LIN {X 0,Y 369.464,Z 431.864,A -85,B 0,C 180,E1 -12702.078,E2 -12702.078} C_VEL
LIN {X 0,Y 369.996,Z 423.683,A -85,B 0,C 180,E1 -12702.896,E2 -12702.896} C_VEL
LIN {X 0,Y 370.537,Z 415.209,A -85,B 0,C 180,E1 -12703.575,E2 -12703.575} C_VEL
LIN {X 0,Y 371.025,Z 406.559,A -85,B 0,C 180,E1 -12704.116,E2 -12704.116} C_VEL
LIN {X 0,Y 371.546,Z 395.482,A -85,B 0,C 180,E1 -12704.62,E2 -12704.62} C_VEL
LIN {X 0,Y 371.88,Z 379.251,A -85,B 0,C 180,E1 -12705.026,E2 -12705.026} C_VEL
LIN {X 0,Y 372.213,Z 341.609,A -85,B 0,C 180,E1 -12705.819,E2 -12705.819} C_VEL
LIN {X 0,Y 369.031,Z 313.014,A -85,B 0,C 180,E1 -12706.559,E2 -12706.559} C_VEL
LIN {X 0,Y 370.022,Z 297.413,A -85,B 0,C 180,E1 -12710.281,E2 -12710.281} C_VEL
LIN {X 0,Y 371.123,Z 283.099,A -85,B 0,C 180,E1 -12713.729,E2 -12713.729} C_VEL
LIN {X 0,Y 370.607,Z 278.235,A -85,B 0,C 180,E1 -12714.957,E2 -12714.957} C_VEL
LIN {X 0,Y 369.016,Z 269.333,A -85,B 0,C 180,E1 -12717.276,E2 -12717.276} C_VEL
LIN {X 0,Y 368.912,Z 269.342,A -85,B 0,C 180,E1 -12720.987,E2 -12720.987} C_VEL
LIN {X 0,Y 368.937,Z 269.338,A -85,B 0,C 180,E1 -12724.853,E2 -12724.853} C_VEL
LIN {X 0,Y 368.909,Z 269.341,A -85,B 0,C 180,E1 -12728.64,E2 -12728.64} C_VEL
LIN {X 0,Y 368.881,Z 269.346,A -85,B 0,C 180,E1 -12732.009,E2 -12732.009} C_VEL
LIN {X 0,Y 368.879,Z 269.347,A -85,B 0,C 180,E1 -12735.175,E2 -12735.175} C_VEL
LIN {X 0,Y 368.881,Z 269.345,A -85,B 0,C 180,E1 -12738.177,E2 -12738.177} C_VEL
LIN {X 0,Y 368.906,Z 269.346,A -85,B 0,C 180,E1 -12741.359,E2 -12741.359} C_VEL
LIN {X 0,Y 368.935,Z 269.34,A -85,B 0,C 180,E1 -12745.146,E2 -12745.146} C_VEL
LIN {X 0,Y 368.928,Z 269.34,A -85,B 0,C 180,E1 -12749.046,E2 -12749.046} C_VEL
LIN {X 0,Y 368.977,Z 269.339,A -85,B 0,C 180,E1 -12751.563,E2 -12751.563} C_VEL
LIN {X 0,Y 368.997,Z 269.332,A -85,B 0,C 180,E1 -12754.019,E2 -12754.019} C_VEL
LIN {X 0,Y 368.929,Z 269.345,A -85,B 0,C 180,E1 -12757.604,E2 -12757.604} C_VEL
LIN {X 0,Y 368.963,Z 269.336,A -85,B 0,C 180,E1 -12761.105,E2 -12761.105} C_VEL
LIN {X 0,Y 368.994,Z 269.33,A -85,B 0,C 180,E1 -12764.534,E2 -12764.534} C_VEL
LIN {X 0,Y 369.001,Z 269.333,A -85,B 0,C 180,E1 -12767.906,E2 -12767.906} C_VEL
LIN {X 0,Y 369.162,Z 269.313,A -85,B 0,C 180,E1 -12771.868,E2 -12771.868} C_VEL
LIN {X 0,Y 369.139,Z 269.313,A -85,B 0,C 180,E1 -12774.537,E2 -12774.537} C_VEL
LIN {X 0,Y 369.313,Z 269.295,A -85,B 0,C 180,E1 -12777.818,E2 -12777.818} C_VEL
LIN {X 0,Y 369.453,Z 269.276,A -85,B 0,C 180,E1 -12779.999,E2 -12779.999} C_VEL
LIN {X 0,Y 369.313,Z 269.292,A -85,B 0,C 180,E1 -12782.18,E2 -12782.18} C_VEL
LIN {X 0,Y 369.197,Z 269.305,A -85,B 0,C 180,E1 -12786.628,E2 -12786.628} C_VEL
LIN {X 0,Y 369.133,Z 269.313,A -85,B 0,C 180,E1 -12788.76,E2 -12788.76} C_VEL
LIN {X 0,Y 369.006,Z 269.331,A -85,B 0,C 180,E1 -12792.092,E2 -12792.092} C_VEL
LIN {X 0,Y 368.992,Z 269.335,A -85,B 0,C 180,E1 -12795.464,E2 -12795.464} C_VEL
LIN {X 0,Y 368.983,Z 269.332,A -85,B 0,C 180,E1 -12798.892,E2 -12798.892} C_VEL
LIN {X 0,Y 368.93,Z 269.339,A -85,B 0,C 180,E1 -12802.394,E2 -12802.394} C_VEL
LIN {X 0,Y 368.992,Z 269.334,A -85,B 0,C 180,E1 -12805.979,E2 -12805.979} C_VEL
LIN {X 0,Y 368.907,Z 269.348,A -85,B 0,C 180,E1 -12809.69,E2 -12809.69} C_VEL
LIN {X 0,Y 368.889,Z 269.345,A -85,B 0,C 180,E1 -12813.042,E2 -12813.042} C_VEL
LIN {X 0,Y 368.91,Z 269.343,A -85,B 0,C 180,E1 -12816.196,E2 -12816.196} C_VEL
LIN {X 0,Y 368.899,Z 269.343,A -85,B 0,C 180,E1 -12818.952,E2 -12818.952} C_VEL
LIN {X 0,Y 368.901,Z 269.345,A -85,B 0,C 180,E1 -12822.014,E2 -12822.014} C_VEL
LIN {X 0,Y 368.946,Z 269.338,A -85,B 0,C 180,E1 -12825.187,E2 -12825.187} C_VEL
LIN {X 0,Y 368.937,Z 269.34,A -85,B 0,C 180,E1 -12828.186,E2 -12828.186} C_VEL
LIN {X 0,Y 368.904,Z 269.345,A -85,B 0,C 180,E1 -12831.358,E2 -12831.358} C_VEL
LIN {X 0,Y 368.928,Z 269.34,A -85,B 0,C 180,E1 -12835.146,E2 -12835.146} C_VEL
LIN {X 0,Y 368.921,Z 269.34,A -85,B 0,C 180,E1 -12839.046,E2 -12839.046} C_VEL
LIN {X 0,Y 368.971,Z 269.338,A -85,B 0,C 180,E1 -12841.564,E2 -12841.564} C_VEL
LIN {X 0,Y 368.991,Z 269.334,A -85,B 0,C 180,E1 -12844.019,E2 -12844.019} C_VEL
LIN {X 0,Y 368.925,Z 269.344,A -85,B 0,C 180,E1 -12847.605,E2 -12847.605} C_VEL
LIN {X 0,Y 368.975,Z 269.334,A -85,B 0,C 180,E1 -12851.107,E2 -12851.107} C_VEL
LIN {X 0,Y 368.989,Z 269.332,A -85,B 0,C 180,E1 -12854.535,E2 -12854.535} C_VEL
LIN {X 0,Y 368.997,Z 269.335,A -85,B 0,C 180,E1 -12857.906,E2 -12857.906} C_VEL
LIN {X 0,Y 369.22,Z 269.308,A -85,B 0,C 180,E1 -12861.801,E2 -12861.801} C_VEL
LIN {X 0,Y 369.133,Z 269.314,A -85,B 0,C 180,E1 -12864.537,E2 -12864.537} C_VEL
LIN {X 0,Y 369.307,Z 269.297,A -85,B 0,C 180,E1 -12867.819,E2 -12867.819} C_VEL
LIN {X 0,Y 369.449,Z 269.278,A -85,B 0,C 180,E1 -12870,E2 -12870} C_VEL
LIN {X 0,Y 369.307,Z 269.294,A -85,B 0,C 180,E1 -12872.181,E2 -12872.181} C_VEL
LIN {X 0,Y 369.189,Z 269.307,A -85,B 0,C 180,E1 -12876.558,E2 -12876.558} C_VEL
LIN {X 0,Y 369.113,Z 269.316,A -85,B 0,C 180,E1 -12878.761,E2 -12878.761} C_VEL
LIN {X 0,Y 369.003,Z 269.333,A -85,B 0,C 180,E1 -12882.093,E2 -12882.093} C_VEL
LIN {X 0,Y 368.989,Z 269.334,A -85,B 0,C 180,E1 -12885.465,E2 -12885.465} C_VEL
LIN {X 0,Y 368.948,Z 269.337,A -85,B 0,C 180,E1 -12888.894,E2 -12888.894} C_VEL
LIN {X 0,Y 368.915,Z 269.342,A -85,B 0,C 180,E1 -12892.395,E2 -12892.395} C_VEL
LIN {X 0,Y 368.989,Z 269.336,A -85,B 0,C 180,E1 -12895.98,E2 -12895.98} C_VEL
LIN {X 0,Y 368.909,Z 269.346,A -85,B 0,C 180,E1 -12899.69,E2 -12899.69} C_VEL
LIN {X 0,Y 368.983,Z 269.414,A -85,B 0,C 180,E1 -12901.322,E2 -12901.322} C_VEL
LIN {X 0,Y 369.531,Z 273.509,A -85,B 0,C 180,E1 -12902.538,E2 -12902.538} C_VEL
LIN {X 0,Y 372.803,Z 292.013,A -85,B 0,C 180,E1 -12903.079,E2 -12903.079} C_VEL
LIN {X 0,Y 372.124,Z 332.295,A -85,B 0,C 180,E1 -12903.917,E2 -12903.917} C_VEL
LIN {X 0,Y 371.303,Z 338.133,A -85,B 0,C 180,E1 -12904.01,E2 -12904.01} C_VEL
LIN {X 0,Y 365.612,Z 355.514,A -85,B 0,C 180,E1 -12904.276,E2 -12904.276} C_VEL
LIN {X 0,Y 364.732,Z 360.703,A -85,B 0,C 180,E1 -12904.47,E2 -12904.47} C_VEL
LIN {X 0,Y 364.647,Z 362.591,A -85,B 0,C 180,E1 -12904.557,E2 -12904.557} C_VEL
LIN {X 0,Y 364.216,Z 373.541,A -85,B 0,C 180,E1 -12905.21,E2 -12905.21} C_VEL
LIN {X 0,Y 363.762,Z 382.837,A -85,B 0,C 180,E1 -12905.955,E2 -12905.955} C_VEL
LIN {X 0,Y 363.399,Z 390.285,A -85,B 0,C 180,E1 -12906.699,E2 -12906.699} C_VEL
LIN {X 0,Y 362.909,Z 397.891,A -85,B 0,C 180,E1 -12907.62,E2 -12907.62} C_VEL
LIN {X 0,Y 362.404,Z 404.176,A -85,B 0,C 180,E1 -12908.532,E2 -12908.532} C_VEL
LIN {X 0,Y 361.95,Z 410.539,A -85,B 0,C 180,E1 -12909.642,E2 -12909.642} C_VEL
LIN {X 0,Y 361.646,Z 415.686,A -85,B 0,C 180,E1 -12910.723,E2 -12910.723} C_VEL
LIN {X 0,Y 361.224,Z 420.228,A -85,B 0,C 180,E1 -12911.862,E2 -12911.862} C_VEL
LIN {X 0,Y 360.948,Z 425.143,A -85,B 0,C 180,E1 -12913.423,E2 -12913.423} C_VEL
LIN {X 0,Y 360.756,Z 427.858,A -85,B 0,C 180,E1 -12914.532,E2 -12914.532} C_VEL
LIN {X 0,Y 360.592,Z 429.716,A -85,B 0,C 180,E1 -12915.443,E2 -12915.443} C_VEL
LIN {X 0,Y 360.403,Z 431.851,A -85,B 0,C 180,E1 -12916.962,E2 -12916.962} C_VEL
LIN {X 0,Y 360.327,Z 433.016,A -85,B 0,C 180,E1 -12918.461,E2 -12918.461} C_VEL
LIN {X 0,Y 360.394,Z 433.266,A -85,B 0,C 180,E1 -12919.946,E2 -12919.946} C_VEL
LIN {X 0,Y 360.52,Z 432.637,A -85,B 0,C 180,E1 -12921.407,E2 -12921.407} C_VEL
LIN {X 0,Y 360.787,Z 430.932,A -85,B 0,C 180,E1 -12923.001,E2 -12923.001} C_VEL
LIN {X 0,Y 361.041,Z 428.802,A -85,B 0,C 180,E1 -12924.271,E2 -12924.271} C_VEL
LIN {X 0,Y 361.424,Z 425.566,A -85,B 0,C 180,E1 -12925.675,E2 -12925.675} C_VEL
LIN {X 0,Y 362.019,Z 420.207,A -85,B 0,C 180,E1 -12927.405,E2 -12927.405} C_VEL
LIN {X 0,Y 362.647,Z 414.276,A -85,B 0,C 180,E1 -12928.862,E2 -12928.862} C_VEL
LIN {X 0,Y 363.301,Z 407.451,A -85,B 0,C 180,E1 -12930.172,E2 -12930.172} C_VEL
LIN {X 0,Y 364.05,Z 400.148,A -85,B 0,C 180,E1 -12931.302,E2 -12931.302} C_VEL
LIN {X 0,Y 364.715,Z 393.335,A -85,B 0,C 180,E1 -12932.174,E2 -12932.174} C_VEL
LIN {X 0,Y 365.239,Z 385.966,A -85,B 0,C 180,E1 -12932.962,E2 -12932.962} C_VEL
LIN {X 0,Y 365.741,Z 377.497,A -85,B 0,C 180,E1 -12933.695,E2 -12933.695} C_VEL
LIN {X 0,Y 366.277,Z 369.067,A -85,B 0,C 180,E1 -12934.264,E2 -12934.264} C_VEL
LIN {X 0,Y 366.592,Z 359.77,A -85,B 0,C 180,E1 -12934.742,E2 -12934.742} C_VEL
LIN {X 0,Y 366.828,Z 350.382,A -85,B 0,C 180,E1 -12935.072,E2 -12935.072} C_VEL
LIN {X 0,Y 367.979,Z 292.659,A -85,B 0,C 180,E1 -12936.356,E2 -12936.356} C_VEL
LIN {X 0,Y 365.505,Z 281.786,A -85,B 0,C 180,E1 -12936.768,E2 -12936.768} C_VEL
LIN {X 0,Y 362.818,Z 274.529,A -85,B 0,C 180,E1 -12937.132,E2 -12937.132} C_VEL
LIN {X 0,Y 361.896,Z 270.225,A -85,B 0,C 180,E1 -12938.349,E2 -12938.349} C_VEL
LIN {X 0,Y 361.957,Z 270.215,A -85,B 0,C 180,E1 -12942.062,E2 -12942.062} C_VEL
LIN {X 0,Y 361.988,Z 270.207,A -85,B 0,C 180,E1 -12946.102,E2 -12946.102} C_VEL
LIN {X 0,Y 362.022,Z 270.202,A -85,B 0,C 180,E1 -12949.939,E2 -12949.939} C_VEL
LIN {X 0,Y 362.158,Z 270.185,A -85,B 0,C 180,E1 -12953.315,E2 -12953.315} C_VEL
LIN {X 0,Y 362.275,Z 270.166,A -85,B 0,C 180,E1 -12957.777,E2 -12957.777} C_VEL
LIN {X 0,Y 362.419,Z 270.153,A -85,B 0,C 180,E1 -12960.001,E2 -12960.001} C_VEL
LIN {X 0,Y 362.275,Z 270.17,A -85,B 0,C 180,E1 -12962.225,E2 -12962.225} C_VEL
LIN {X 0,Y 362.164,Z 270.185,A -85,B 0,C 180,E1 -12966.687,E2 -12966.687} C_VEL
LIN {X 0,Y 362.067,Z 270.194,A -85,B 0,C 180,E1 -12968.934,E2 -12968.934} C_VEL
LIN {X 0,Y 361.952,Z 270.205,A -85,B 0,C 180,E1 -12972.333,E2 -12972.333} C_VEL
LIN {X 0,Y 361.955,Z 270.212,A -85,B 0,C 180,E1 -12974.621,E2 -12974.621} C_VEL
LIN {X 0,Y 361.953,Z 270.207,A -85,B 0,C 180,E1 -12978.1,E2 -12978.1} C_VEL
LIN {X 0,Y 361.886,Z 270.211,A -85,B 0,C 180,E1 -12981.654,E2 -12981.654} C_VEL
LIN {X 0,Y 361.923,Z 270.205,A -85,B 0,C 180,E1 -12985.291,E2 -12985.291} C_VEL
LIN {X 0,Y 361.917,Z 270.214,A -85,B 0,C 180,E1 -12987.779,E2 -12987.779} C_VEL
LIN {X 0,Y 361.842,Z 270.223,A -85,B 0,C 180,E1 -12991.286,E2 -12991.286} C_VEL
LIN {X 0,Y 361.85,Z 270.218,A -85,B 0,C 180,E1 -12994.282,E2 -12994.282} C_VEL
LIN {X 0,Y 361.862,Z 270.216,A -85,B 0,C 180,E1 -12997.224,E2 -12997.224} C_VEL
LIN {X 0,Y 361.87,Z 270.218,A -85,B 0,C 180,E1 -13000.763,E2 -13000.763} C_VEL
LIN {X 0,Y 361.861,Z 270.22,A -85,B 0,C 180,E1 -13004.362,E2 -13004.362} C_VEL
LIN {X 0,Y 361.834,Z 270.225,A -85,B 0,C 180,E1 -13007.569,E2 -13007.569} C_VEL
LIN {X 0,Y 361.869,Z 270.221,A -85,B 0,C 180,E1 -13010.974,E2 -13010.974} C_VEL
LIN {X 0,Y 361.873,Z 270.223,A -85,B 0,C 180,E1 -13014.656,E2 -13014.656} C_VEL
LIN {X 0,Y 361.837,Z 270.228,A -85,B 0,C 180,E1 -13018.372,E2 -13018.372} C_VEL
LIN {X 0,Y 361.918,Z 270.267,A -85,B 0,C 180,E1 -13022.183,E2 -13022.183} C_VEL
LIN {X 0,Y 363.78,Z 279.211,A -85,B 0,C 180,E1 -13024.542,E2 -13024.542} C_VEL
LIN {X 0,Y 364.457,Z 284.393,A -85,B 0,C 180,E1 -13025.849,E2 -13025.849} C_VEL
LIN {X 0,Y 363.322,Z 299.23,A -85,B 0,C 180,E1 -13029.328,E2 -13029.328} C_VEL
LIN {X 0,Y 362.603,Z 310.337,A -85,B 0,C 180,E1 -13031.912,E2 -13031.912} C_VEL
LIN {X 0,Y 366.013,Z 332.015,A -85,B 0,C 180,E1 -13032.637,E2 -13032.637} C_VEL
LIN {X 0,Y 367.237,Z 345.692,A -85,B 0,C 180,E1 -13033.023,E2 -13033.023} C_VEL
LIN {X 0,Y 366.326,Z 389.941,A -85,B 0,C 180,E1 -13034.016,E2 -13034.016} C_VEL
LIN {X 0,Y 365.823,Z 401.663,A -85,B 0,C 180,E1 -13034.47,E2 -13034.47} C_VEL
LIN {X 0,Y 365.072,Z 412.017,A -85,B 0,C 180,E1 -13035.08,E2 -13035.08} C_VEL
LIN {X 0,Y 364.371,Z 420.792,A -85,B 0,C 180,E1 -13035.764,E2 -13035.764} C_VEL
LIN {X 0,Y 363.598,Z 429.21,A -85,B 0,C 180,E1 -13036.589,E2 -13036.589} C_VEL
LIN {X 0,Y 362.832,Z 437.203,A -85,B 0,C 180,E1 -13037.556,E2 -13037.556} C_VEL
LIN {X 0,Y 362.272,Z 443.836,A -85,B 0,C 180,E1 -13038.531,E2 -13038.531} C_VEL
LIN {X 0,Y 361.636,Z 450.167,A -85,B 0,C 180,E1 -13039.645,E2 -13039.645} C_VEL
LIN {X 0,Y 361.155,Z 455.45,A -85,B 0,C 180,E1 -13040.762,E2 -13040.762} C_VEL
LIN {X 0,Y 360.783,Z 460.854,A -85,B 0,C 180,E1 -13042.163,E2 -13042.163} C_VEL
LIN {X 0,Y 360.496,Z 465.95,A -85,B 0,C 180,E1 -13043.863,E2 -13043.863} C_VEL
LIN {X 0,Y 360.451,Z 469.439,A -85,B 0,C 180,E1 -13045.527,E2 -13045.527} C_VEL
LIN {X 0,Y 360.376,Z 471.138,A -85,B 0,C 180,E1 -13046.646,E2 -13046.646} C_VEL
LIN {X 0,Y 360.426,Z 472.224,A -85,B 0,C 180,E1 -13047.765,E2 -13047.765} C_VEL
LIN {X 0,Y 360.513,Z 472.804,A -85,B 0,C 180,E1 -13048.883,E2 -13048.883} C_VEL
LIN {X 0,Y 360.515,Z 472.899,A -85,B 0,C 180,E1 -13050,E2 -13050} C_VEL
LIN {X 0,Y 360.522,Z 472.509,A -85,B 0,C 180,E1 -13051.117,E2 -13051.117} C_VEL
LIN {X 0,Y 360.47,Z 471.553,A -85,B 0,C 180,E1 -13052.235,E2 -13052.235} C_VEL
LIN {X 0,Y 360.434,Z 469.062,A -85,B 0,C 180,E1 -13053.913,E2 -13053.913} C_VEL
LIN {X 0,Y 360.475,Z 466.715,A -85,B 0,C 180,E1 -13055.033,E2 -13055.033} C_VEL
LIN {X 0,Y 360.582,Z 461.895,A -85,B 0,C 180,E1 -13056.716,E2 -13056.716} C_VEL
LIN {X 0,Y 360.8,Z 456.651,A -85,B 0,C 180,E1 -13058.119,E2 -13058.119} C_VEL
LIN {X 0,Y 361.108,Z 451.511,A -85,B 0,C 180,E1 -13059.24,E2 -13059.24} C_VEL
LIN {X 0,Y 361.499,Z 445.309,A -85,B 0,C 180,E1 -13060.36,E2 -13060.36} C_VEL
LIN {X 0,Y 361.896,Z 438.787,A -85,B 0,C 180,E1 -13061.34,E2 -13061.34} C_VEL
LIN {X 0,Y 362.509,Z 430.909,A -85,B 0,C 180,E1 -13062.313,E2 -13062.313} C_VEL
LIN {X 0,Y 363.057,Z 422.603,A -85,B 0,C 180,E1 -13063.147,E2 -13063.147} C_VEL
LIN {X 0,Y 363.66,Z 412.069,A -85,B 0,C 180,E1 -13063.979,E2 -13063.979} C_VEL
LIN {X 0,Y 364.264,Z 400.977,A -85,B 0,C 180,E1 -13064.593,E2 -13064.593} C_VEL
LIN {X 0,Y 364.685,Z 391.599,A -85,B 0,C 180,E1 -13064.947,E2 -13064.947} C_VEL
LIN {X 0,Y 365.233,Z 356.793,A -85,B 0,C 180,E1 -13065.725,E2 -13065.725} C_VEL
LIN {X 0,Y 365.323,Z 342.507,A -85,B 0,C 180,E1 -13066.035,E2 -13066.035} C_VEL
LIN {X 0,Y 362.032,Z 312.562,A -85,B 0,C 180,E1 -13066.849,E2 -13066.849} C_VEL
LIN {X 0,Y 362.985,Z 298.012,A -85,B 0,C 180,E1 -13070.396,E2 -13070.396} C_VEL
LIN {X 0,Y 364.132,Z 283.685,A -85,B 0,C 180,E1 -13073.911,E2 -13073.911} C_VEL
LIN {X 0,Y 363.095,Z 276.349,A -85,B 0,C 180,E1 -13075.817,E2 -13075.817} C_VEL
LIN {X 0,Y 361.958,Z 270.213,A -85,B 0,C 180,E1 -13077.454,E2 -13077.454} C_VEL
LIN {X 0,Y 361.848,Z 270.224,A -85,B 0,C 180,E1 -13081.285,E2 -13081.285} C_VEL
LIN {X 0,Y 361.855,Z 270.22,A -85,B 0,C 180,E1 -13084.28,E2 -13084.28} C_VEL
LIN {X 0,Y 361.871,Z 270.221,A -85,B 0,C 180,E1 -13087.224,E2 -13087.224} C_VEL
LIN {X 0,Y 361.836,Z 270.222,A -85,B 0,C 180,E1 -13090.755,E2 -13090.755} C_VEL
LIN {X 0,Y 361.816,Z 270.225,A -85,B 0,C 180,E1 -13094.368,E2 -13094.368} C_VEL
LIN {X 0,Y 361.835,Z 270.229,A -85,B 0,C 180,E1 -13097.567,E2 -13097.567} C_VEL
LIN {X 0,Y 361.867,Z 270.219,A -85,B 0,C 180,E1 -13100.973,E2 -13100.973} C_VEL
LIN {X 0,Y 361.873,Z 270.217,A -85,B 0,C 180,E1 -13104.654,E2 -13104.654} C_VEL
LIN {X 0,Y 361.837,Z 270.222,A -85,B 0,C 180,E1 -13108.37,E2 -13108.37} C_VEL
LIN {X 0,Y 361.899,Z 270.215,A -85,B 0,C 180,E1 -13110.954,E2 -13110.954} C_VEL
LIN {X 0,Y 361.952,Z 270.213,A -85,B 0,C 180,E1 -13113.474,E2 -13113.474} C_VEL
LIN {X 0,Y 361.887,Z 270.218,A -85,B 0,C 180,E1 -13117.144,E2 -13117.144} C_VEL
LIN {X 0,Y 361.908,Z 270.213,A -85,B 0,C 180,E1 -13120.723,E2 -13120.723} C_VEL
LIN {X 0,Y 361.93,Z 270.212,A -85,B 0,C 180,E1 -13123.065,E2 -13123.065} C_VEL
LIN {X 0,Y 361.995,Z 270.202,A -85,B 0,C 180,E1 -13126.527,E2 -13126.527} C_VEL
LIN {X 0,Y 362.027,Z 270.201,A -85,B 0,C 180,E1 -13129.937,E2 -13129.937} C_VEL
LIN {X 0,Y 362.158,Z 270.185,A -85,B 0,C 180,E1 -13133.313,E2 -13133.313} C_VEL
LIN {X 0,Y 362.277,Z 270.172,A -85,B 0,C 180,E1 -13137.776,E2 -13137.776} C_VEL
LIN {X 0,Y 362.422,Z 270.152,A -85,B 0,C 180,E1 -13139.999,E2 -13139.999} C_VEL
LIN {X 0,Y 362.277,Z 270.168,A -85,B 0,C 180,E1 -13142.223,E2 -13142.223} C_VEL
LIN {X 0,Y 362.166,Z 270.181,A -85,B 0,C 180,E1 -13146.685,E2 -13146.685} C_VEL
LIN {X 0,Y 362.07,Z 270.194,A -85,B 0,C 180,E1 -13148.932,E2 -13148.932} C_VEL
LIN {X 0,Y 361.96,Z 270.208,A -85,B 0,C 180,E1 -13152.331,E2 -13152.331} C_VEL
LIN {X 0,Y 361.956,Z 270.207,A -85,B 0,C 180,E1 -13154.619,E2 -13154.619} C_VEL
LIN {X 0,Y 361.954,Z 270.21,A -85,B 0,C 180,E1 -13158.098,E2 -13158.098} C_VEL
LIN {X 0,Y 361.892,Z 270.222,A -85,B 0,C 180,E1 -13161.652,E2 -13161.652} C_VEL
LIN {X 0,Y 361.921,Z 270.214,A -85,B 0,C 180,E1 -13165.289,E2 -13165.289} C_VEL
LIN {X 0,Y 361.9,Z 270.219,A -85,B 0,C 180,E1 -13167.778,E2 -13167.778} C_VEL
LIN {X 0,Y 361.83,Z 270.229,A -85,B 0,C 180,E1 -13171.629,E2 -13171.629} C_VEL
LIN {X 0,Y 361.866,Z 270.221,A -85,B 0,C 180,E1 -13175.344,E2 -13175.344} C_VEL
LIN {X 0,Y 361.866,Z 270.219,A -85,B 0,C 180,E1 -13179.027,E2 -13179.027} C_VEL
LIN {X 0,Y 361.849,Z 270.221,A -85,B 0,C 180,E1 -13182.435,E2 -13182.435} C_VEL
LIN {X 0,Y 361.903,Z 270.218,A -85,B 0,C 180,E1 -13185.931,E2 -13185.931} C_VEL
LIN {X 0,Y 361.898,Z 270.216,A -85,B 0,C 180,E1 -13189.231,E2 -13189.231} C_VEL
LIN {X 0,Y 361.86,Z 270.22,A -85,B 0,C 180,E1 -13192.982,E2 -13192.982} C_VEL
LIN {X 0,Y 361.85,Z 270.221,A -85,B 0,C 180,E1 -13196.63,E2 -13196.63} C_VEL
LIN {X 0,Y 361.866,Z 270.224,A -85,B 0,C 180,E1 -13199.672,E2 -13199.672} C_VEL
LIN {X 0,Y 361.946,Z 270.212,A -85,B 0,C 180,E1 -13203.475,E2 -13203.475} C_VEL
LIN {X 0,Y 361.882,Z 270.218,A -85,B 0,C 180,E1 -13207.144,E2 -13207.144} C_VEL
LIN {X 0,Y 361.913,Z 270.213,A -85,B 0,C 180,E1 -13210.724,E2 -13210.724} C_VEL
LIN {X 0,Y 361.937,Z 270.212,A -85,B 0,C 180,E1 -13214.226,E2 -13214.226} C_VEL
LIN {X 0,Y 361.99,Z 270.204,A -85,B 0,C 180,E1 -13216.528,E2 -13216.528} C_VEL
LIN {X 0,Y 362.023,Z 270.203,A -85,B 0,C 180,E1 -13219.938,E2 -13219.938} C_VEL
LIN {X 0,Y 362.142,Z 270.187,A -85,B 0,C 180,E1 -13222.192,E2 -13222.192} C_VEL
LIN {X 0,Y 362.107,Z 270.19,A -85,B 0,C 180,E1 -13224.431,E2 -13224.431} C_VEL
LIN {X 0,Y 362.271,Z 270.174,A -85,B 0,C 180,E1 -13227.776,E2 -13227.776} C_VEL
LIN {X 0,Y 362.419,Z 270.154,A -85,B 0,C 180,E1 -13230,E2 -13230} C_VEL
LIN {X 0,Y 362.271,Z 270.171,A -85,B 0,C 180,E1 -13232.223,E2 -13232.223} C_VEL
LIN {X 0,Y 362.151,Z 270.183,A -85,B 0,C 180,E1 -13236.686,E2 -13236.686} C_VEL
LIN {X 0,Y 362.026,Z 270.202,A -85,B 0,C 180,E1 -13240.062,E2 -13240.062} C_VEL
LIN {X 0,Y 361.989,Z 270.208,A -85,B 0,C 180,E1 -13243.899,E2 -13243.899} C_VEL
LIN {X 0,Y 361.958,Z 270.212,A -85,B 0,C 180,E1 -13247.938,E2 -13247.938} C_VEL
LIN {X 0,Y 361.871,Z 270.223,A -85,B 0,C 180,E1 -13251.653,E2 -13251.653} C_VEL
LIN {X 0,Y 361.916,Z 270.214,A -85,B 0,C 180,E1 -13255.29,E2 -13255.29} C_VEL
LIN {X 0,Y 361.897,Z 270.221,A -85,B 0,C 180,E1 -13257.779,E2 -13257.779} C_VEL
LIN {X 0,Y 361.959,Z 270.345,A -85,B 0,C 180,E1 -13261.207,E2 -13261.207} C_VEL
LIN {X 0,Y 362.487,Z 273.827,A -85,B 0,C 180,E1 -13262.26,E2 -13262.26} C_VEL
LIN {X 0,Y 365.894,Z 292.494,A -85,B 0,C 180,E1 -13262.83,E2 -13262.83} C_VEL
LIN {X 0,Y 364.927,Z 351.352,A -85,B 0,C 180,E1 -13264.119,E2 -13264.119} C_VEL
LIN {X 0,Y 364.654,Z 361.835,A -85,B 0,C 180,E1 -13264.521,E2 -13264.521} C_VEL
LIN {X 0,Y 364.647,Z 362.591,A -85,B 0,C 180,E1 -13264.557,E2 -13264.557} C_VEL
LIN {X 0,Y 363.888,Z 368.188,A -85,B 0,C 180,E1 -13264.83,E2 -13264.83} C_VEL
LIN {X 0,Y 360.708,Z 377.043,A -85,B 0,C 180,E1 -13265.331,E2 -13265.331} C_VEL
LIN {X 0,Y 357.4,Z 385.465,A -85,B 0,C 180,E1 -13265.981,E2 -13265.981} C_VEL
LIN {X 0,Y 356.447,Z 390.376,A -85,B 0,C 180,E1 -13266.485,E2 -13266.485} C_VEL
LIN {X 0,Y 355.947,Z 397.73,A -85,B 0,C 180,E1 -13267.382,E2 -13267.382} C_VEL
LIN {X 0,Y 355.4,Z 404.322,A -85,B 0,C 180,E1 -13268.346,E2 -13268.346} C_VEL
LIN {X 0,Y 354.939,Z 410.577,A -85,B 0,C 180,E1 -13269.448,E2 -13269.448} C_VEL
LIN {X 0,Y 354.632,Z 415.496,A -85,B 0,C 180,E1 -13270.48,E2 -13270.48} C_VEL
LIN {X 0,Y 354.174,Z 420.483,A -85,B 0,C 180,E1 -13271.74,E2 -13271.74} C_VEL
LIN {X 0,Y 353.997,Z 423.786,A -85,B 0,C 180,E1 -13272.731,E2 -13272.731} C_VEL
LIN {X 0,Y 353.706,Z 427.903,A -85,B 0,C 180,E1 -13274.334,E2 -13274.334} C_VEL
LIN {X 0,Y 353.441,Z 430.805,A -85,B 0,C 180,E1 -13275.898,E2 -13275.898} C_VEL
LIN {X 0,Y 353.272,Z 432.663,A -85,B 0,C 180,E1 -13277.439,E2 -13277.439} C_VEL
LIN {X 0,Y 353.266,Z 433.615,A -85,B 0,C 180,E1 -13279.11,E2 -13279.11} C_VEL
LIN {X 0,Y 353.377,Z 433.471,A -85,B 0,C 180,E1 -13280.861,E2 -13280.861} C_VEL
LIN {X 0,Y 353.643,Z 432.029,A -85,B 0,C 180,E1 -13282.646,E2 -13282.646} C_VEL
LIN {X 0,Y 354.032,Z 429.137,A -85,B 0,C 180,E1 -13284.477,E2 -13284.477} C_VEL
LIN {X 0,Y 354.586,Z 424.715,A -85,B 0,C 180,E1 -13286.349,E2 -13286.349} C_VEL
LIN {X 0,Y 355.224,Z 419.162,A -85,B 0,C 180,E1 -13288.037,E2 -13288.037} C_VEL
LIN {X 0,Y 355.827,Z 413.335,A -85,B 0,C 180,E1 -13289.397,E2 -13289.397} C_VEL
LIN {X 0,Y 356.548,Z 406.736,A -85,B 0,C 180,E1 -13290.64,E2 -13290.64} C_VEL
LIN {X 0,Y 357.284,Z 400.061,A -85,B 0,C 180,E1 -13291.671,E2 -13291.671} C_VEL
LIN {X 0,Y 357.942,Z 393.314,A -85,B 0,C 180,E1 -13292.54,E2 -13292.54} C_VEL
LIN {X 0,Y 358.516,Z 385.817,A -85,B 0,C 180,E1 -13293.345,E2 -13293.345} C_VEL
LIN {X 0,Y 359.023,Z 377.786,A -85,B 0,C 180,E1 -13294.047,E2 -13294.047} C_VEL
LIN {X 0,Y 359.56,Z 369.575,A -85,B 0,C 180,E1 -13294.61,E2 -13294.61} C_VEL
LIN {X 0,Y 359.927,Z 359.785,A -85,B 0,C 180,E1 -13295.121,E2 -13295.121} C_VEL
LIN {X 0,Y 360.21,Z 349.811,A -85,B 0,C 180,E1 -13295.468,E2 -13295.468} C_VEL
LIN {X 0,Y 361.42,Z 294.009,A -85,B 0,C 180,E1 -13296.736,E2 -13296.736} C_VEL
LIN {X 0,Y 359.237,Z 284.276,A -85,B 0,C 180,E1 -13297.114,E2 -13297.114} C_VEL
LIN {X 0,Y 355.654,Z 274.96,A -85,B 0,C 180,E1 -13297.605,E2 -13297.605} C_VEL
LIN {X 0,Y 354.831,Z 271.105,A -85,B 0,C 180,E1 -13298.714,E2 -13298.714} C_VEL
LIN {X 0,Y 354.913,Z 271.092,A -85,B 0,C 180,E1 -13301.892,E2 -13301.892} C_VEL
LIN {X 0,Y 354.933,Z 271.086,A -85,B 0,C 180,E1 -13305.982,E2 -13305.982} C_VEL
LIN {X 0,Y 354.969,Z 271.081,A -85,B 0,C 180,E1 -13309.737,E2 -13309.737} C_VEL
LIN {X 0,Y 355.12,Z 271.063,A -85,B 0,C 180,E1 -13313.181,E2 -13313.181} C_VEL
LIN {X 0,Y 355.238,Z 271.043,A -85,B 0,C 180,E1 -13317.733,E2 -13317.733} C_VEL
LIN {X 0,Y 355.389,Z 271.029,A -85,B 0,C 180,E1 -13320.001,E2 -13320.001} C_VEL
LIN {X 0,Y 355.238,Z 271.047,A -85,B 0,C 180,E1 -13322.269,E2 -13322.269} C_VEL
LIN {X 0,Y 355.13,Z 271.06,A -85,B 0,C 180,E1 -13326.82,E2 -13326.82} C_VEL
LIN {X 0,Y 355.008,Z 271.074,A -85,B 0,C 180,E1 -13329.113,E2 -13329.113} C_VEL
LIN {X 0,Y 354.913,Z 271.082,A -85,B 0,C 180,E1 -13332.582,E2 -13332.582} C_VEL
LIN {X 0,Y 354.883,Z 271.087,A -85,B 0,C 180,E1 -13336.097,E2 -13336.097} C_VEL
LIN {X 0,Y 354.9,Z 271.089,A -85,B 0,C 180,E1 -13338.473,E2 -13338.473} C_VEL
LIN {X 0,Y 354.829,Z 271.092,A -85,B 0,C 180,E1 -13342.107,E2 -13342.107} C_VEL
LIN {X 0,Y 354.894,Z 271.081,A -85,B 0,C 180,E1 -13345.829,E2 -13345.829} C_VEL
LIN {X 0,Y 354.85,Z 271.086,A -85,B 0,C 180,E1 -13349.68,E2 -13349.68} C_VEL
LIN {X 0,Y 354.802,Z 271.092,A -85,B 0,C 180,E1 -13353.703,E2 -13353.703} C_VEL
LIN {X 0,Y 354.796,Z 271.1,A -85,B 0,C 180,E1 -13356.46,E2 -13356.46} C_VEL
LIN {X 0,Y 354.821,Z 271.098,A -85,B 0,C 180,E1 -13359.425,E2 -13359.425} C_VEL
LIN {X 0,Y 354.802,Z 271.1,A -85,B 0,C 180,E1 -13362.871,E2 -13362.871} C_VEL
LIN {X 0,Y 354.766,Z 271.106,A -85,B 0,C 180,E1 -13366.105,E2 -13366.105} C_VEL
LIN {X 0,Y 354.786,Z 271.102,A -85,B 0,C 180,E1 -13369.18,E2 -13369.18} C_VEL
LIN {X 0,Y 354.811,Z 271.105,A -85,B 0,C 180,E1 -13372.403,E2 -13372.403} C_VEL
LIN {X 0,Y 354.811,Z 271.101,A -85,B 0,C 180,E1 -13374.942,E2 -13374.942} C_VEL
LIN {X 0,Y 354.793,Z 271.106,A -85,B 0,C 180,E1 -13378.406,E2 -13378.406} C_VEL
LIN {X 0,Y 354.896,Z 271.146,A -85,B 0,C 180,E1 -13381.825,E2 -13381.825} C_VEL
LIN {X 0,Y 357.069,Z 281.772,A -85,B 0,C 180,E1 -13384.686,E2 -13384.686} C_VEL
LIN {X 0,Y 357.533,Z 286.656,A -85,B 0,C 180,E1 -13385.929,E2 -13385.929} C_VEL
LIN {X 0,Y 356.166,Z 302.865,A -85,B 0,C 180,E1 -13389.8,E2 -13389.8} C_VEL
LIN {X 0,Y 355.693,Z 309.903,A -85,B 0,C 180,E1 -13391.464,E2 -13391.464} C_VEL
LIN {X 0,Y 359.216,Z 331.764,A -85,B 0,C 180,E1 -13392.224,E2 -13392.224} C_VEL
LIN {X 0,Y 360.554,Z 345.594,A -85,B 0,C 180,E1 -13392.637,E2 -13392.637} C_VEL
LIN {X 0,Y 359.634,Z 389.254,A -85,B 0,C 180,E1 -13393.638,E2 -13393.638} C_VEL
LIN {X 0,Y 359.125,Z 400.506,A -85,B 0,C 180,E1 -13394.073,E2 -13394.073} C_VEL
LIN {X 0,Y 358.227,Z 412.409,A -85,B 0,C 180,E1 -13394.788,E2 -13394.788} C_VEL
LIN {X 0,Y 357.517,Z 421.027,A -85,B 0,C 180,E1 -13395.485,E2 -13395.485} C_VEL
LIN {X 0,Y 356.71,Z 429.331,A -85,B 0,C 180,E1 -13396.325,E2 -13396.325} C_VEL
LIN {X 0,Y 355.906,Z 437.239,A -85,B 0,C 180,E1 -13397.31,E2 -13397.31} C_VEL
LIN {X 0,Y 355.282,Z 443.801,A -85,B 0,C 180,E1 -13398.302,E2 -13398.302} C_VEL
LIN {X 0,Y 354.642,Z 450.073,A -85,B 0,C 180,E1 -13399.438,E2 -13399.438} C_VEL
LIN {X 0,Y 354.02,Z 456.503,A -85,B 0,C 180,E1 -13400.862,E2 -13400.862} C_VEL
LIN {X 0,Y 353.629,Z 462.497,A -85,B 0,C 180,E1 -13402.578,E2 -13402.578} C_VEL
LIN {X 0,Y 353.335,Z 466.877,A -85,B 0,C 180,E1 -13404.293,E2 -13404.293} C_VEL
LIN {X 0,Y 353.358,Z 469.113,A -85,B 0,C 180,E1 -13405.437,E2 -13405.437} C_VEL
LIN {X 0,Y 353.296,Z 470.8,A -85,B 0,C 180,E1 -13406.579,E2 -13406.579} C_VEL
LIN {X 0,Y 353.327,Z 471.873,A -85,B 0,C 180,E1 -13407.72,E2 -13407.72} C_VEL
LIN {X 0,Y 353.429,Z 472.424,A -85,B 0,C 180,E1 -13408.861,E2 -13408.861} C_VEL
LIN {X 0,Y 353.451,Z 472.486,A -85,B 0,C 180,E1 -13410,E2 -13410} C_VEL
LIN {X 0,Y 353.458,Z 472.064,A -85,B 0,C 180,E1 -13411.14,E2 -13411.14} C_VEL
LIN {X 0,Y 353.374,Z 471.097,A -85,B 0,C 180,E1 -13412.28,E2 -13412.28} C_VEL
LIN {X 0,Y 353.364,Z 468.545,A -85,B 0,C 180,E1 -13413.992,E2 -13413.992} C_VEL
LIN {X 0,Y 353.369,Z 466.175,A -85,B 0,C 180,E1 -13415.135,E2 -13415.135} C_VEL
LIN {X 0,Y 353.519,Z 461.29,A -85,B 0,C 180,E1 -13416.851,E2 -13416.851} C_VEL
LIN {X 0,Y 353.756,Z 455.996,A -85,B 0,C 180,E1 -13418.281,E2 -13418.281} C_VEL
LIN {X 0,Y 354.039,Z 450.794,A -85,B 0,C 180,E1 -13419.426,E2 -13419.426} C_VEL
LIN {X 0,Y 354.501,Z 444.53,A -85,B 0,C 180,E1 -13420.567,E2 -13420.567} C_VEL
LIN {X 0,Y 354.922,Z 437.929,A -85,B 0,C 180,E1 -13421.566,E2 -13421.566} C_VEL
LIN {X 0,Y 355.545,Z 429.952,A -85,B 0,C 180,E1 -13422.558,E2 -13422.558} C_VEL
LIN {X 0,Y 356.249,Z 420.017,A -85,B 0,C 180,E1 -13423.548,E2 -13423.548} C_VEL
LIN {X 0,Y 356.834,Z 409.546,A -85,B 0,C 180,E1 -13424.325,E2 -13424.325} C_VEL
LIN {X 0,Y 357.381,Z 399.216,A -85,B 0,C 180,E1 -13424.876,E2 -13424.876} C_VEL
LIN {X 0,Y 357.775,Z 390.076,A -85,B 0,C 180,E1 -13425.21,E2 -13425.21} C_VEL
LIN {X 0,Y 358.432,Z 343.387,A -85,B 0,C 180,E1 -13426.261,E2 -13426.261} C_VEL
LIN {X 0,Y 354.98,Z 312.274,A -85,B 0,C 180,E1 -13427.113,E2 -13427.113} C_VEL
LIN {X 0,Y 355.964,Z 298.575,A -85,B 0,C 180,E1 -13430.515,E2 -13430.515} C_VEL
LIN {X 0,Y 357.068,Z 285.463,A -85,B 0,C 180,E1 -13433.796,E2 -13433.796} C_VEL
LIN {X 0,Y 356.682,Z 280.896,A -85,B 0,C 180,E1 -13434.99,E2 -13434.99} C_VEL
LIN {X 0,Y 354.91,Z 271.091,A -85,B 0,C 180,E1 -13437.644,E2 -13437.644} C_VEL
LIN {X 0,Y 354.795,Z 271.105,A -85,B 0,C 180,E1 -13441.594,E2 -13441.594} C_VEL
LIN {X 0,Y 354.813,Z 271.099,A -85,B 0,C 180,E1 -13445.059,E2 -13445.059} C_VEL
LIN {X 0,Y 354.809,Z 271.1,A -85,B 0,C 180,E1 -13447.882,E2 -13447.882} C_VEL
LIN {X 0,Y 354.788,Z 271.102,A -85,B 0,C 180,E1 -13451.171,E2 -13451.171} C_VEL
LIN {X 0,Y 354.763,Z 271.103,A -85,B 0,C 180,E1 -13454.505,E2 -13454.505} C_VEL
LIN {X 0,Y 354.793,Z 271.105,A -85,B 0,C 180,E1 -13457.662,E2 -13457.662} C_VEL
LIN {X 0,Y 354.815,Z 271.097,A -85,B 0,C 180,E1 -13460.665,E2 -13460.665} C_VEL
LIN {X 0,Y 354.82,Z 271.096,A -85,B 0,C 180,E1 -13464.3,E2 -13464.3} C_VEL
LIN {X 0,Y 354.787,Z 271.106,A -85,B 0,C 180,E1 -13467.666,E2 -13467.666} C_VEL
LIN {X 0,Y 354.867,Z 271.09,A -85,B 0,C 180,E1 -13470.62,E2 -13470.62} C_VEL
LIN {X 0,Y 354.897,Z 271.088,A -85,B 0,C 180,E1 -13474.172,E2 -13474.172} C_VEL
LIN {X 0,Y 354.832,Z 271.098,A -85,B 0,C 180,E1 -13477.893,E2 -13477.893} C_VEL
LIN {X 0,Y 354.92,Z 271.087,A -85,B 0,C 180,E1 -13481.891,E2 -13481.891} C_VEL
LIN {X 0,Y 354.939,Z 271.084,A -85,B 0,C 180,E1 -13485.98,E2 -13485.98} C_VEL
LIN {X 0,Y 354.974,Z 271.082,A -85,B 0,C 180,E1 -13489.735,E2 -13489.735} C_VEL
LIN {X 0,Y 355.121,Z 271.061,A -85,B 0,C 180,E1 -13493.18,E2 -13493.18} C_VEL
LIN {X 0,Y 355.241,Z 271.049,A -85,B 0,C 180,E1 -13497.731,E2 -13497.731} C_VEL
LIN {X 0,Y 355.392,Z 271.028,A -85,B 0,C 180,E1 -13499.999,E2 -13499.999} C_VEL
LIN {X 0,Y 355.24,Z 271.045,A -85,B 0,C 180,E1 -13502.267,E2 -13502.267} C_VEL
LIN {X 0,Y 355.132,Z 271.057,A -85,B 0,C 180,E1 -13506.818,E2 -13506.818} C_VEL
LIN {X 0,Y 355.011,Z 271.074,A -85,B 0,C 180,E1 -13509.111,E2 -13509.111} C_VEL
LIN {X 0,Y 354.919,Z 271.084,A -85,B 0,C 180,E1 -13512.58,E2 -13512.58} C_VEL
LIN {X 0,Y 354.883,Z 271.091,A -85,B 0,C 180,E1 -13516.095,E2 -13516.095} C_VEL
LIN {X 0,Y 354.902,Z 271.086,A -85,B 0,C 180,E1 -13518.471,E2 -13518.471} C_VEL
LIN {X 0,Y 354.832,Z 271.097,A -85,B 0,C 180,E1 -13522.105,E2 -13522.105} C_VEL
LIN {X 0,Y 354.892,Z 271.092,A -85,B 0,C 180,E1 -13525.827,E2 -13525.827} C_VEL
LIN {X 0,Y 354.838,Z 271.1,A -85,B 0,C 180,E1 -13529.679,E2 -13529.679} C_VEL
LIN {X 0,Y 354.798,Z 271.105,A -85,B 0,C 180,E1 -13533.701,E2 -13533.701} C_VEL
LIN {X 0,Y 354.793,Z 271.1,A -85,B 0,C 180,E1 -13536.458,E2 -13536.458} C_VEL
LIN {X 0,Y 354.816,Z 271.1,A -85,B 0,C 180,E1 -13539.423,E2 -13539.423} C_VEL
LIN {X 0,Y 354.8,Z 271.099,A -85,B 0,C 180,E1 -13542.87,E2 -13542.87} C_VEL
LIN {X 0,Y 354.843,Z 271.096,A -85,B 0,C 180,E1 -13546.116,E2 -13546.116} C_VEL
LIN {X 0,Y 354.849,Z 271.094,A -85,B 0,C 180,E1 -13549.188,E2 -13549.188} C_VEL
LIN {X 0,Y 354.8,Z 271.099,A -85,B 0,C 180,E1 -13552.402,E2 -13552.402} C_VEL
LIN {X 0,Y 354.803,Z 271.099,A -85,B 0,C 180,E1 -13554.94,E2 -13554.94} C_VEL
LIN {X 0,Y 354.784,Z 271.102,A -85,B 0,C 180,E1 -13558.405,E2 -13558.405} C_VEL
LIN {X 0,Y 354.842,Z 271.098,A -85,B 0,C 180,E1 -13561.619,E2 -13561.619} C_VEL
LIN {X 0,Y 354.891,Z 271.09,A -85,B 0,C 180,E1 -13564.172,E2 -13564.172} C_VEL
LIN {X 0,Y 354.827,Z 271.1,A -85,B 0,C 180,E1 -13567.894,E2 -13567.894} C_VEL
LIN {X 0,Y 354.915,Z 271.089,A -85,B 0,C 180,E1 -13571.891,E2 -13571.891} C_VEL
LIN {X 0,Y 354.934,Z 271.086,A -85,B 0,C 180,E1 -13575.981,E2 -13575.981} C_VEL
LIN {X 0,Y 354.97,Z 271.084,A -85,B 0,C 180,E1 -13579.736,E2 -13579.736} C_VEL
LIN {X 0,Y 355.105,Z 271.064,A -85,B 0,C 180,E1 -13582.037,E2 -13582.037} C_VEL
LIN {X 0,Y 355.081,Z 271.065,A -85,B 0,C 180,E1 -13584.32,E2 -13584.32} C_VEL
LIN {X 0,Y 355.234,Z 271.051,A -85,B 0,C 180,E1 -13587.732,E2 -13587.732} C_VEL
LIN {X 0,Y 355.388,Z 271.03,A -85,B 0,C 180,E1 -13590,E2 -13590} C_VEL
LIN {X 0,Y 355.235,Z 271.047,A -85,B 0,C 180,E1 -13592.267,E2 -13592.267} C_VEL
LIN {X 0,Y 355.116,Z 271.06,A -85,B 0,C 180,E1 -13596.819,E2 -13596.819} C_VEL
LIN {X 0,Y 354.973,Z 271.079,A -85,B 0,C 180,E1 -13600.264,E2 -13600.264} C_VEL
LIN {X 0,Y 354.934,Z 271.086,A -85,B 0,C 180,E1 -13604.019,E2 -13604.019} C_VEL
LIN {X 0,Y 354.913,Z 271.088,A -85,B 0,C 180,E1 -13608.108,E2 -13608.108} C_VEL
LIN {X 0,Y 354.817,Z 271.1,A -85,B 0,C 180,E1 -13612.106,E2 -13612.106} C_VEL
LIN {X 0,Y 354.888,Z 271.094,A -85,B 0,C 180,E1 -13615.827,E2 -13615.827} C_VEL
LIN {X 0,Y 354.844,Z 271.098,A -85,B 0,C 180,E1 -13619.678,E2 -13619.678} C_VEL
LIN {X 0,Y 354.903,Z 271.151,A -85,B 0,C 180,E1 -13621.044,E2 -13621.044} C_VEL
LIN {X 0,Y 355.394,Z 274.239,A -85,B 0,C 180,E1 -13621.999,E2 -13621.999} C_VEL
LIN {X 0,Y 358.994,Z 293.2,A -85,B 0,C 180,E1 -13622.576,E2 -13622.576} C_VEL
LIN {X 0,Y 358.016,Z 351.095,A -85,B 0,C 180,E1 -13623.87,E2 -13623.87} C_VEL
LIN {X 0,Y 357.71,Z 361.094,A -85,B 0,C 180,E1 -13624.247,E2 -13624.247} C_VEL
LIN {X 0,Y 357.398,Z 371.896,A -85,B 0,C 180,E1 -13624.853,E2 -13624.853} C_VEL
LIN {X 0,Y 356.813,Z 382.552,A -85,B 0,C 180,E1 -13625.697,E2 -13625.697} C_VEL
LIN {X 0,Y 356.447,Z 390.376,A -85,B 0,C 180,E1 -13626.485,E2 -13626.485} C_VEL
LIN {X 0,Y 355.501,Z 395.253,A -85,B 0,C 180,E1 -13627.027,E2 -13627.027} C_VEL
LIN {X 0,Y 352.079,Z 402.669,A -85,B 0,C 180,E1 -13627.971,E2 -13627.971} C_VEL
LIN {X 0,Y 348.698,Z 409.346,A -85,B 0,C 180,E1 -13629.022,E2 -13629.022} C_VEL
LIN {X 0,Y 347.767,Z 413.018,A -85,B 0,C 180,E1 -13629.742,E2 -13629.742} C_VEL
LIN {X 0,Y 347.175,Z 420.306,A -85,B 0,C 180,E1 -13631.498,E2 -13631.498} C_VEL
LIN {X 0,Y 346.966,Z 423.772,A -85,B 0,C 180,E1 -13632.536,E2 -13632.536} C_VEL
LIN {X 0,Y 346.66,Z 428.022,A -85,B 0,C 180,E1 -13634.178,E2 -13634.178} C_VEL
LIN {X 0,Y 346.473,Z 430.168,A -85,B 0,C 180,E1 -13635.23,E2 -13635.23} C_VEL
LIN {X 0,Y 346.213,Z 432.594,A -85,B 0,C 180,E1 -13636.951,E2 -13636.951} C_VEL
LIN {X 0,Y 346.168,Z 433.855,A -85,B 0,C 180,E1 -13638.691,E2 -13638.691} C_VEL
LIN {X 0,Y 346.196,Z 434.118,A -85,B 0,C 180,E1 -13639.489,E2 -13639.489} C_VEL
LIN {X 0,Y 346.305,Z 433.862,A -85,B 0,C 180,E1 -13641.016,E2 -13641.016} C_VEL
LIN {X 0,Y 346.534,Z 432.736,A -85,B 0,C 180,E1 -13642.526,E2 -13642.526} C_VEL
LIN {X 0,Y 346.888,Z 430.552,A -85,B 0,C 180,E1 -13644.133,E2 -13644.133} C_VEL
LIN {X 0,Y 347.269,Z 427.889,A -85,B 0,C 180,E1 -13645.484,E2 -13645.484} C_VEL
LIN {X 0,Y 347.725,Z 424.107,A -85,B 0,C 180,E1 -13646.929,E2 -13646.929} C_VEL
LIN {X 0,Y 348.288,Z 419.278,A -85,B 0,C 180,E1 -13648.357,E2 -13648.357} C_VEL
LIN {X 0,Y 348.982,Z 413.242,A -85,B 0,C 180,E1 -13649.772,E2 -13649.772} C_VEL
LIN {X 0,Y 349.759,Z 406.736,A -85,B 0,C 180,E1 -13651.004,E2 -13651.004} C_VEL
LIN {X 0,Y 350.537,Z 399.713,A -85,B 0,C 180,E1 -13652.097,E2 -13652.097} C_VEL
LIN {X 0,Y 351.3,Z 391.938,A -85,B 0,C 180,E1 -13653.089,E2 -13653.089} C_VEL
LIN {X 0,Y 352.092,Z 382.046,A -85,B 0,C 180,E1 -13654.102,E2 -13654.102} C_VEL
LIN {X 0,Y 352.77,Z 371.836,A -85,B 0,C 180,E1 -13654.876,E2 -13654.876} C_VEL
LIN {X 0,Y 353.186,Z 361.599,A -85,B 0,C 180,E1 -13655.448,E2 -13655.448} C_VEL
LIN {X 0,Y 353.491,Z 352.572,A -85,B 0,C 180,E1 -13655.794,E2 -13655.794} C_VEL
LIN {X 0,Y 354.738,Z 294.652,A -85,B 0,C 180,E1 -13657.16,E2 -13657.16} C_VEL
LIN {X 0,Y 352.837,Z 286.37,A -85,B 0,C 180,E1 -13657.493,E2 -13657.493} C_VEL
LIN {X 0,Y 348.571,Z 275.424,A -85,B 0,C 180,E1 -13658.103,E2 -13658.103} C_VEL
LIN {X 0,Y 347.78,Z 271.985,A -85,B 0,C 180,E1 -13659.136,E2 -13659.136} C_VEL
LIN {X 0,Y 347.856,Z 271.972,A -85,B 0,C 180,E1 -13662.36,E2 -13662.36} C_VEL
LIN {X 0,Y 347.888,Z 271.963,A -85,B 0,C 180,E1 -13665.972,E2 -13665.972} C_VEL
LIN {X 0,Y 347.919,Z 271.959,A -85,B 0,C 180,E1 -13669.526,E2 -13669.526} C_VEL
LIN {X 0,Y 348.086,Z 271.94,A -85,B 0,C 180,E1 -13673.043,E2 -13673.043} C_VEL
LIN {X 0,Y 348.2,Z 271.919,A -85,B 0,C 180,E1 -13677.687,E2 -13677.687} C_VEL
LIN {X 0,Y 348.338,Z 271.908,A -85,B 0,C 180,E1 -13680.001,E2 -13680.001} C_VEL
LIN {X 0,Y 348.2,Z 271.924,A -85,B 0,C 180,E1 -13682.314,E2 -13682.314} C_VEL
LIN {X 0,Y 348.098,Z 271.935,A -85,B 0,C 180,E1 -13686.959,E2 -13686.959} C_VEL
LIN {X 0,Y 347.96,Z 271.951,A -85,B 0,C 180,E1 -13689.3,E2 -13689.3} C_VEL
LIN {X 0,Y 347.882,Z 271.958,A -85,B 0,C 180,E1 -13692.841,E2 -13692.841} C_VEL
LIN {X 0,Y 347.832,Z 271.963,A -85,B 0,C 180,E1 -13696.433,E2 -13696.433} C_VEL
LIN {X 0,Y 347.85,Z 271.967,A -85,B 0,C 180,E1 -13698.861,E2 -13698.861} C_VEL
LIN {X 0,Y 347.768,Z 271.977,A -85,B 0,C 180,E1 -13702.581,E2 -13702.581} C_VEL
LIN {X 0,Y 347.807,Z 271.963,A -85,B 0,C 180,E1 -13705.11,E2 -13705.11} C_VEL
LIN {X 0,Y 347.807,Z 271.971,A -85,B 0,C 180,E1 -13707.695,E2 -13707.695} C_VEL
LIN {X 0,Y 347.76,Z 271.973,A -85,B 0,C 180,E1 -13710.348,E2 -13710.348} C_VEL
LIN {X 0,Y 347.741,Z 271.978,A -85,B 0,C 180,E1 -13714.465,E2 -13714.465} C_VEL
LIN {X 0,Y 347.773,Z 271.972,A -85,B 0,C 180,E1 -13717.99,E2 -13717.99} C_VEL
LIN {X 0,Y 347.764,Z 271.977,A -85,B 0,C 180,E1 -13721.829,E2 -13721.829} C_VEL
LIN {X 0,Y 347.765,Z 271.979,A -85,B 0,C 180,E1 -13725.018,E2 -13725.018} C_VEL
LIN {X 0,Y 347.748,Z 271.982,A -85,B 0,C 180,E1 -13728.398,E2 -13728.398} C_VEL
LIN {X 0,Y 347.776,Z 271.978,A -85,B 0,C 180,E1 -13732.012,E2 -13732.012} C_VEL
LIN {X 0,Y 347.744,Z 271.981,A -85,B 0,C 180,E1 -13735.537,E2 -13735.537} C_VEL
LIN {X 0,Y 347.745,Z 271.983,A -85,B 0,C 180,E1 -13738.301,E2 -13738.301} C_VEL
LIN {X 0,Y 347.842,Z 272.09,A -85,B 0,C 180,E1 -13741.448,E2 -13741.448} C_VEL
LIN {X 0,Y 349.632,Z 280.355,A -85,B 0,C 180,E1 -13743.755,E2 -13743.755} C_VEL
LIN {X 0,Y 350.63,Z 286.621,A -85,B 0,C 180,E1 -13745.424,E2 -13745.424} C_VEL
LIN {X 0,Y 349.742,Z 297.829,A -85,B 0,C 180,E1 -13748.177,E2 -13748.177} C_VEL
LIN {X 0,Y 348.835,Z 309.651,A -85,B 0,C 180,E1 -13750.997,E2 -13750.997} C_VEL
LIN {X 0,Y 352.551,Z 332.016,A -85,B 0,C 180,E1 -13751.805,E2 -13751.805} C_VEL
LIN {X 0,Y 353.921,Z 345.911,A -85,B 0,C 180,E1 -13752.233,E2 -13752.233} C_VEL
LIN {X 0,Y 352.948,Z 388.728,A -85,B 0,C 180,E1 -13753.242,E2 -13753.242} C_VEL
LIN {X 0,Y 352.435,Z 399.74,A -85,B 0,C 180,E1 -13753.675,E2 -13753.675} C_VEL
LIN {X 0,Y 351.63,Z 410.971,A -85,B 0,C 180,E1 -13754.347,E2 -13754.347} C_VEL
LIN {X 0,Y 350.667,Z 421.266,A -85,B 0,C 180,E1 -13755.195,E2 -13755.195} C_VEL
LIN {X 0,Y 349.834,Z 429.458,A -85,B 0,C 180,E1 -13756.051,E2 -13756.051} C_VEL
LIN {X 0,Y 348.99,Z 437.28,A -85,B 0,C 180,E1 -13757.054,E2 -13757.054} C_VEL
LIN {X 0,Y 348.128,Z 445.511,A -85,B 0,C 180,E1 -13758.354,E2 -13758.354} C_VEL
LIN {X 0,Y 347.354,Z 452.741,A -85,B 0,C 180,E1 -13759.803,E2 -13759.803} C_VEL
LIN {X 0,Y 346.831,Z 458.48,A -85,B 0,C 180,E1 -13761.259,E2 -13761.259} C_VEL
LIN {X 0,Y 346.441,Z 463.847,A -85,B 0,C 180,E1 -13763.009,E2 -13763.009} C_VEL
LIN {X 0,Y 346.225,Z 467.822,A -85,B 0,C 180,E1 -13764.759,E2 -13764.759} C_VEL
LIN {X 0,Y 346.217,Z 470.466,A -85,B 0,C 180,E1 -13766.509,E2 -13766.509} C_VEL
LIN {X 0,Y 346.229,Z 471.528,A -85,B 0,C 180,E1 -13767.674,E2 -13767.674} C_VEL
LIN {X 0,Y 346.347,Z 472.043,A -85,B 0,C 180,E1 -13768.838,E2 -13768.838} C_VEL
LIN {X 0,Y 346.388,Z 472.073,A -85,B 0,C 180,E1 -13770,E2 -13770} C_VEL
LIN {X 0,Y 346.375,Z 471.615,A -85,B 0,C 180,E1 -13771.163,E2 -13771.163} C_VEL
LIN {X 0,Y 346.278,Z 470.632,A -85,B 0,C 180,E1 -13772.327,E2 -13772.327} C_VEL
LIN {X 0,Y 346.296,Z 468.025,A -85,B 0,C 180,E1 -13774.073,E2 -13774.073} C_VEL
LIN {X 0,Y 346.268,Z 465.627,A -85,B 0,C 180,E1 -13775.241,E2 -13775.241} C_VEL
LIN {X 0,Y 346.442,Z 460.682,A -85,B 0,C 180,E1 -13776.991,E2 -13776.991} C_VEL
LIN {X 0,Y 346.723,Z 455.339,A -85,B 0,C 180,E1 -13778.451,E2 -13778.451} C_VEL
LIN {X 0,Y 346.989,Z 450.074,A -85,B 0,C 180,E1 -13779.619,E2 -13779.619} C_VEL
LIN {X 0,Y 347.51,Z 443.747,A -85,B 0,C 180,E1 -13780.782,E2 -13780.782} C_VEL
LIN {X 0,Y 348.085,Z 436.039,A -85,B 0,C 180,E1 -13781.944,E2 -13781.944} C_VEL
LIN {X 0,Y 348.742,Z 426.426,A -85,B 0,C 180,E1 -13783.104,E2 -13783.104} C_VEL
LIN {X 0,Y 349.438,Z 417.055,A -85,B 0,C 180,E1 -13783.966,E2 -13783.966} C_VEL
LIN {X 0,Y 349.95,Z 408.046,A -85,B 0,C 180,E1 -13784.613,E2 -13784.613} C_VEL
LIN {X 0,Y 350.493,Z 398.109,A -85,B 0,C 180,E1 -13785.14,E2 -13785.14} C_VEL
LIN {X 0,Y 350.879,Z 388.649,A -85,B 0,C 180,E1 -13785.48,E2 -13785.48} C_VEL
LIN {X 0,Y 351.437,Z 343.15,A -85,B 0,C 180,E1 -13786.527,E2 -13786.527} C_VEL
LIN {X 0,Y 347.986,Z 311.859,A -85,B 0,C 180,E1 -13787.407,E2 -13787.407} C_VEL
LIN {X 0,Y 348.928,Z 299.132,A -85,B 0,C 180,E1 -13790.639,E2 -13790.639} C_VEL
LIN {X 0,Y 350.077,Z 286.015,A -85,B 0,C 180,E1 -13793.987,E2 -13793.987} C_VEL
LIN {X 0,Y 349.573,Z 281.43,A -85,B 0,C 180,E1 -13795.216,E2 -13795.216} C_VEL
LIN {X 0,Y 347.876,Z 271.966,A -85,B 0,C 180,E1 -13797.851,E2 -13797.851} C_VEL
LIN {X 0,Y 347.74,Z 271.98,A -85,B 0,C 180,E1 -13801.913,E2 -13801.913} C_VEL
LIN {X 0,Y 347.79,Z 271.975,A -85,B 0,C 180,E1 -13805.875,E2 -13805.875} C_VEL
LIN {X 0,Y 347.754,Z 271.977,A -85,B 0,C 180,E1 -13808.792,E2 -13808.792} C_VEL
LIN {X 0,Y 347.751,Z 271.98,A -85,B 0,C 180,E1 -13811.83,E2 -13811.83} C_VEL
LIN {X 0,Y 347.705,Z 271.984,A -85,B 0,C 180,E1 -13815.026,E2 -13815.026} C_VEL
LIN {X 0,Y 347.749,Z 271.977,A -85,B 0,C 180,E1 -13818.396,E2 -13818.396} C_VEL
LIN {X 0,Y 347.772,Z 271.976,A -85,B 0,C 180,E1 -13822.011,E2 -13822.011} C_VEL
LIN {X 0,Y 347.743,Z 271.984,A -85,B 0,C 180,E1 -13825.535,E2 -13825.535} C_VEL
LIN {X 0,Y 347.762,Z 271.981,A -85,B 0,C 180,E1 -13829.653,E2 -13829.653} C_VEL
LIN {X 0,Y 347.85,Z 271.964,A -85,B 0,C 180,E1 -13832.744,E2 -13832.744} C_VEL
LIN {X 0,Y 347.786,Z 271.974,A -85,B 0,C 180,E1 -13836.161,E2 -13836.161} C_VEL
LIN {X 0,Y 347.811,Z 271.972,A -85,B 0,C 180,E1 -13839.908,E2 -13839.908} C_VEL
LIN {X 0,Y 347.863,Z 271.963,A -85,B 0,C 180,E1 -13842.358,E2 -13842.358} C_VEL
LIN {X 0,Y 347.894,Z 271.962,A -85,B 0,C 180,E1 -13845.97,E2 -13845.97} C_VEL
LIN {X 0,Y 347.924,Z 271.96,A -85,B 0,C 180,E1 -13849.525,E2 -13849.525} C_VEL
LIN {X 0,Y 348.087,Z 271.936,A -85,B 0,C 180,E1 -13853.041,E2 -13853.041} C_VEL
LIN {X 0,Y 348.203,Z 271.926,A -85,B 0,C 180,E1 -13857.686,E2 -13857.686} C_VEL
LIN {X 0,Y 348.341,Z 271.906,A -85,B 0,C 180,E1 -13859.999,E2 -13859.999} C_VEL
LIN {X 0,Y 348.203,Z 271.921,A -85,B 0,C 180,E1 -13862.312,E2 -13862.312} C_VEL
LIN {X 0,Y 348.1,Z 271.934,A -85,B 0,C 180,E1 -13866.957,E2 -13866.957} C_VEL
LIN {X 0,Y 347.963,Z 271.953,A -85,B 0,C 180,E1 -13869.298,E2 -13869.298} C_VEL
LIN {X 0,Y 347.887,Z 271.96,A -85,B 0,C 180,E1 -13872.838,E2 -13872.838} C_VEL
LIN {X 0,Y 347.833,Z 271.967,A -85,B 0,C 180,E1 -13876.43,E2 -13876.43} C_VEL
LIN {X 0,Y 347.853,Z 271.964,A -85,B 0,C 180,E1 -13878.859,E2 -13878.859} C_VEL
LIN {X 0,Y 347.77,Z 271.974,A -85,B 0,C 180,E1 -13882.578,E2 -13882.578} C_VEL
LIN {X 0,Y 347.805,Z 271.971,A -85,B 0,C 180,E1 -13885.108,E2 -13885.108} C_VEL
LIN {X 0,Y 347.801,Z 271.977,A -85,B 0,C 180,E1 -13887.693,E2 -13887.693} C_VEL
LIN {X 0,Y 347.753,Z 271.977,A -85,B 0,C 180,E1 -13890.346,E2 -13890.346} C_VEL
LIN {X 0,Y 347.736,Z 271.979,A -85,B 0,C 180,E1 -13894.463,E2 -13894.463} C_VEL
LIN {X 0,Y 347.771,Z 271.978,A -85,B 0,C 180,E1 -13897.989,E2 -13897.989} C_VEL
LIN {X 0,Y 347.759,Z 271.981,A -85,B 0,C 180,E1 -13901.827,E2 -13901.827} C_VEL
LIN {X 0,Y 347.791,Z 271.972,A -85,B 0,C 180,E1 -13905.011,E2 -13905.011} C_VEL
LIN {X 0,Y 347.778,Z 271.974,A -85,B 0,C 180,E1 -13908.39,E2 -13908.39} C_VEL
LIN {X 0,Y 347.768,Z 271.978,A -85,B 0,C 180,E1 -13912.01,E2 -13912.01} C_VEL
LIN {X 0,Y 347.736,Z 271.983,A -85,B 0,C 180,E1 -13915.536,E2 -13915.536} C_VEL
LIN {X 0,Y 347.755,Z 271.982,A -85,B 0,C 180,E1 -13919.653,E2 -13919.653} C_VEL
LIN {X 0,Y 347.843,Z 271.965,A -85,B 0,C 180,E1 -13922.744,E2 -13922.744} C_VEL
LIN {X 0,Y 347.78,Z 271.976,A -85,B 0,C 180,E1 -13926.162,E2 -13926.162} C_VEL
LIN {X 0,Y 347.81,Z 271.974,A -85,B 0,C 180,E1 -13929.909,E2 -13929.909} C_VEL
LIN {X 0,Y 347.858,Z 271.965,A -85,B 0,C 180,E1 -13932.359,E2 -13932.359} C_VEL
LIN {X 0,Y 347.889,Z 271.964,A -85,B 0,C 180,E1 -13935.97,E2 -13935.97} C_VEL
LIN {X 0,Y 347.92,Z 271.959,A -85,B 0,C 180,E1 -13939.525,E2 -13939.525} C_VEL
LIN {X 0,Y 348.065,Z 271.943,A -85,B 0,C 180,E1 -13941.874,E2 -13941.874} C_VEL
LIN {X 0,Y 348.057,Z 271.941,A -85,B 0,C 180,E1 -13944.205,E2 -13944.205} C_VEL
LIN {X 0,Y 348.196,Z 271.927,A -85,B 0,C 180,E1 -13947.686,E2 -13947.686} C_VEL
LIN {X 0,Y 348.337,Z 271.908,A -85,B 0,C 180,E1 -13950,E2 -13950} C_VEL
LIN {X 0,Y 348.197,Z 271.923,A -85,B 0,C 180,E1 -13952.313,E2 -13952.313} C_VEL
LIN {X 0,Y 348.082,Z 271.936,A -85,B 0,C 180,E1 -13956.958,E2 -13956.958} C_VEL
LIN {X 0,Y 347.923,Z 271.956,A -85,B 0,C 180,E1 -13960.474,E2 -13960.474} C_VEL
LIN {X 0,Y 347.889,Z 271.963,A -85,B 0,C 180,E1 -13964.15,E2 -13964.15} C_VEL
LIN {X 0,Y 347.881,Z 271.963,A -85,B 0,C 180,E1 -13968.29,E2 -13968.29} C_VEL
LIN {X 0,Y 347.766,Z 271.979,A -85,B 0,C 180,E1 -13971.63,E2 -13971.63} C_VEL
LIN {X 0,Y 347.801,Z 271.971,A -85,B 0,C 180,E1 -13975.108,E2 -13975.108} C_VEL
LIN {X 0,Y 347.798,Z 271.976,A -85,B 0,C 180,E1 -13977.694,E2 -13977.694} C_VEL
LIN {X 0,Y 347.848,Z 272.126,A -85,B 0,C 180,E1 -13980.926,E2 -13980.926} C_VEL
LIN {X 0,Y 348.339,Z 274.831,A -85,B 0,C 180,E1 -13981.72,E2 -13981.72} C_VEL
LIN {X 0,Y 350.96,Z 287.268,A -85,B 0,C 180,E1 -13982.121,E2 -13982.121} C_VEL
LIN {X 0,Y 352.098,Z 293.857,A -85,B 0,C 180,E1 -13982.32,E2 -13982.32} C_VEL
LIN {X 0,Y 351.086,Z 351.395,A -85,B 0,C 180,E1 -13983.636,E2 -13983.636} C_VEL
LIN {X 0,Y 350.773,Z 361.284,A -85,B 0,C 180,E1 -13984.016,E2 -13984.016} C_VEL
LIN {X 0,Y 350.391,Z 372.834,A -85,B 0,C 180,E1 -13984.681,E2 -13984.681} C_VEL
LIN {X 0,Y 349.822,Z 383.028,A -85,B 0,C 180,E1 -13985.511,E2 -13985.511} C_VEL
LIN {X 0,Y 349.382,Z 391.814,A -85,B 0,C 180,E1 -13986.429,E2 -13986.429} C_VEL
LIN {X 0,Y 348.827,Z 399.448,A -85,B 0,C 180,E1 -13987.407,E2 -13987.407} C_VEL
LIN {X 0,Y 348.202,Z 406.882,A -85,B 0,C 180,E1 -13988.569,E2 -13988.569} C_VEL
LIN {X 0,Y 347.767,Z 413.018,A -85,B 0,C 180,E1 -13989.742,E2 -13989.742} C_VEL
LIN {X 0,Y 346.863,Z 416.6,A -85,B 0,C 180,E1 -13990.502,E2 -13990.502} C_VEL
LIN {X 0,Y 343.589,Z 421.761,A -85,B 0,C 180,E1 -13991.8,E2 -13991.8} C_VEL
LIN {X 0,Y 340.373,Z 426.084,A -85,B 0,C 180,E1 -13993.205,E2 -13993.205} C_VEL
LIN {X 0,Y 339.579,Z 428.324,A -85,B 0,C 180,E1 -13994.12,E2 -13994.12} C_VEL
LIN {X 0,Y 339.372,Z 430.6,A -85,B 0,C 180,E1 -13995.245,E2 -13995.245} C_VEL
LIN {X 0,Y 339.139,Z 432.878,A -85,B 0,C 180,E1 -13996.856,E2 -13996.856} C_VEL
LIN {X 0,Y 339.078,Z 434.158,A -85,B 0,C 180,E1 -13998.453,E2 -13998.453} C_VEL
LIN {X 0,Y 339.148,Z 434.507,A -85,B 0,C 180,E1 -14000.06,E2 -14000.06} C_VEL
LIN {X 0,Y 339.346,Z 433.74,A -85,B 0,C 180,E1 -14001.904,E2 -14001.904} C_VEL
LIN {X 0,Y 339.711,Z 431.711,A -85,B 0,C 180,E1 -14003.786,E2 -14003.786} C_VEL
LIN {X 0,Y 340.266,Z 428.257,A -85,B 0,C 180,E1 -14005.706,E2 -14005.706} C_VEL
LIN {X 0,Y 340.789,Z 424.321,A -85,B 0,C 180,E1 -14007.226,E2 -14007.226} C_VEL
LIN {X 0,Y 341.391,Z 419.373,A -85,B 0,C 180,E1 -14008.705,E2 -14008.705} C_VEL
LIN {X 0,Y 342.104,Z 413.586,A -85,B 0,C 180,E1 -14010.085,E2 -14010.085} C_VEL
LIN {X 0,Y 342.817,Z 408.144,A -85,B 0,C 180,E1 -14011.153,E2 -14011.153} C_VEL
LIN {X 0,Y 343.633,Z 401.27,A -85,B 0,C 180,E1 -14012.273,E2 -14012.273} C_VEL
LIN {X 0,Y 344.463,Z 393.332,A -85,B 0,C 180,E1 -14013.331,E2 -14013.331} C_VEL
LIN {X 0,Y 345.225,Z 384.664,A -85,B 0,C 180,E1 -14014.264,E2 -14014.264} C_VEL
LIN {X 0,Y 345.961,Z 374.389,A -85,B 0,C 180,E1 -14015.13,E2 -14015.13} C_VEL
LIN {X 0,Y 346.526,Z 363.473,A -85,B 0,C 180,E1 -14015.781,E2 -14015.781} C_VEL
LIN {X 0,Y 346.867,Z 353.564,A -85,B 0,C 180,E1 -14016.185,E2 -14016.185} C_VEL
LIN {X 0,Y 348.217,Z 295.886,A -85,B 0,C 180,E1 -14017.578,E2 -14017.578} C_VEL
LIN {X 0,Y 346.634,Z 288.921,A -85,B 0,C 180,E1 -14017.872,E2 -14017.872} C_VEL
LIN {X 0,Y 341.399,Z 275.824,A -85,B 0,C 180,E1 -14018.648,E2 -14018.648} C_VEL
LIN {X 0,Y 340.768,Z 272.857,A -85,B 0,C 180,E1 -14019.556,E2 -14019.556} C_VEL
LIN {X 0,Y 340.848,Z 272.844,A -85,B 0,C 180,E1 -14021.985,E2 -14021.985} C_VEL
LIN {X 0,Y 340.86,Z 272.839,A -85,B 0,C 180,E1 -14025.706,E2 -14025.706} C_VEL
LIN {X 0,Y 340.862,Z 272.839,A -85,B 0,C 180,E1 -14029.307,E2 -14029.307} C_VEL
LIN {X 0,Y 341.053,Z 272.816,A -85,B 0,C 180,E1 -14032.899,E2 -14032.899} C_VEL
LIN {X 0,Y 341.162,Z 272.796,A -85,B 0,C 180,E1 -14037.64,E2 -14037.64} C_VEL
LIN {X 0,Y 341.288,Z 272.786,A -85,B 0,C 180,E1 -14040.001,E2 -14040.001} C_VEL
LIN {X 0,Y 341.162,Z 272.801,A -85,B 0,C 180,E1 -14042.362,E2 -14042.362} C_VEL
LIN {X 0,Y 341.068,Z 272.809,A -85,B 0,C 180,E1 -14047.103,E2 -14047.103} C_VEL
LIN {X 0,Y 340.863,Z 272.838,A -85,B 0,C 180,E1 -14050.695,E2 -14050.695} C_VEL
LIN {X 0,Y 340.857,Z 272.839,A -85,B 0,C 180,E1 -14054.326,E2 -14054.326} C_VEL
LIN {X 0,Y 340.832,Z 272.841,A -85,B 0,C 180,E1 -14058.468,E2 -14058.468} C_VEL
LIN {X 0,Y 340.748,Z 272.844,A -85,B 0,C 180,E1 -14061.858,E2 -14061.858} C_VEL
LIN {X 0,Y 340.768,Z 272.84,A -85,B 0,C 180,E1 -14065.666,E2 -14065.666} C_VEL
LIN {X 0,Y 340.738,Z 272.851,A -85,B 0,C 180,E1 -14068.321,E2 -14068.321} C_VEL
LIN {X 0,Y 340.7,Z 272.858,A -85,B 0,C 180,E1 -14071.045,E2 -14071.045} C_VEL
LIN {X 0,Y 340.715,Z 272.856,A -85,B 0,C 180,E1 -14075.28,E2 -14075.28} C_VEL
LIN {X 0,Y 340.715,Z 272.855,A -85,B 0,C 180,E1 -14078.389,E2 -14078.389} C_VEL
LIN {X 0,Y 340.73,Z 272.854,A -85,B 0,C 180,E1 -14082.053,E2 -14082.053} C_VEL
LIN {X 0,Y 340.681,Z 272.86,A -85,B 0,C 180,E1 -14085.463,E2 -14085.463} C_VEL
LIN {X 0,Y 340.684,Z 272.86,A -85,B 0,C 180,E1 -14088.692,E2 -14088.692} C_VEL
LIN {X 0,Y 340.734,Z 272.854,A -85,B 0,C 180,E1 -14091.774,E2 -14091.774} C_VEL
LIN {X 0,Y 340.722,Z 272.856,A -85,B 0,C 180,E1 -14095.597,E2 -14095.597} C_VEL
LIN {X 0,Y 340.698,Z 272.861,A -85,B 0,C 180,E1 -14098.956,E2 -14098.956} C_VEL
LIN {X 0,Y 340.766,Z 272.905,A -85,B 0,C 180,E1 -14101.01,E2 -14101.01} C_VEL
LIN {X 0,Y 342.668,Z 281.573,A -85,B 0,C 180,E1 -14103.499,E2 -14103.499} C_VEL
LIN {X 0,Y 343.703,Z 287.831,A -85,B 0,C 180,E1 -14105.218,E2 -14105.218} C_VEL
LIN {X 0,Y 343.242,Z 294.058,A -85,B 0,C 180,E1 -14106.788,E2 -14106.788} C_VEL
LIN {X 0,Y 341.968,Z 309.164,A -85,B 0,C 180,E1 -14110.492,E2 -14110.492} C_VEL
LIN {X 0,Y 345.839,Z 331.913,A -85,B 0,C 180,E1 -14111.357,E2 -14111.357} C_VEL
LIN {X 0,Y 347.326,Z 346.419,A -85,B 0,C 180,E1 -14111.819,E2 -14111.819} C_VEL
LIN {X 0,Y 346.28,Z 389.232,A -85,B 0,C 180,E1 -14112.856,E2 -14112.856} C_VEL
LIN {X 0,Y 345.683,Z 400.917,A -85,B 0,C 180,E1 -14113.348,E2 -14113.348} C_VEL
LIN {X 0,Y 344.805,Z 411.555,A -85,B 0,C 180,E1 -14114.029,E2 -14114.029} C_VEL
LIN {X 0,Y 343.989,Z 420.153,A -85,B 0,C 180,E1 -14114.75,E2 -14114.75} C_VEL
LIN {X 0,Y 343.079,Z 428.446,A -85,B 0,C 180,E1 -14115.619,E2 -14115.619} C_VEL
LIN {X 0,Y 342.151,Z 436.347,A -85,B 0,C 180,E1 -14116.64,E2 -14116.64} C_VEL
LIN {X 0,Y 341.364,Z 443.774,A -85,B 0,C 180,E1 -14117.818,E2 -14117.818} C_VEL
LIN {X 0,Y 340.498,Z 451.342,A -85,B 0,C 180,E1 -14119.295,E2 -14119.295} C_VEL
LIN {X 0,Y 339.862,Z 457.301,A -85,B 0,C 180,E1 -14120.778,E2 -14120.778} C_VEL
LIN {X 0,Y 339.508,Z 462.035,A -85,B 0,C 180,E1 -14122.268,E2 -14122.268} C_VEL
LIN {X 0,Y 339.3,Z 465.125,A -85,B 0,C 180,E1 -14123.459,E2 -14123.459} C_VEL
LIN {X 0,Y 339.157,Z 468.497,A -85,B 0,C 180,E1 -14125.246,E2 -14125.246} C_VEL
LIN {X 0,Y 339.14,Z 470.129,A -85,B 0,C 180,E1 -14126.436,E2 -14126.436} C_VEL
LIN {X 0,Y 339.134,Z 471.185,A -85,B 0,C 180,E1 -14127.625,E2 -14127.625} C_VEL
LIN {X 0,Y 339.251,Z 471.664,A -85,B 0,C 180,E1 -14128.813,E2 -14128.813} C_VEL
LIN {X 0,Y 339.326,Z 471.655,A -85,B 0,C 180,E1 -14130,E2 -14130} C_VEL
LIN {X 0,Y 339.295,Z 471.155,A -85,B 0,C 180,E1 -14131.187,E2 -14131.187} C_VEL
LIN {X 0,Y 339.185,Z 470.145,A -85,B 0,C 180,E1 -14132.375,E2 -14132.375} C_VEL
LIN {X 0,Y 339.227,Z 467.478,A -85,B 0,C 180,E1 -14134.158,E2 -14134.158} C_VEL
LIN {X 0,Y 339.246,Z 463.182,A -85,B 0,C 180,E1 -14136.066,E2 -14136.066} C_VEL
LIN {X 0,Y 339.475,Z 458.078,A -85,B 0,C 180,E1 -14137.734,E2 -14137.734} C_VEL
LIN {X 0,Y 339.809,Z 452.164,A -85,B 0,C 180,E1 -14139.224,E2 -14139.224} C_VEL
LIN {X 0,Y 340.376,Z 444.606,A -85,B 0,C 180,E1 -14140.71,E2 -14140.71} C_VEL
LIN {X 0,Y 340.885,Z 437.133,A -85,B 0,C 180,E1 -14141.898,E2 -14141.898} C_VEL
LIN {X 0,Y 341.56,Z 429.151,A -85,B 0,C 180,E1 -14142.93,E2 -14142.93} C_VEL
LIN {X 0,Y 342.283,Z 419.202,A -85,B 0,C 180,E1 -14143.961,E2 -14143.961} C_VEL
LIN {X 0,Y 342.921,Z 408.707,A -85,B 0,C 180,E1 -14144.768,E2 -14144.768} C_VEL
LIN {X 0,Y 343.526,Z 398.181,A -85,B 0,C 180,E1 -14145.348,E2 -14145.348} C_VEL
LIN {X 0,Y 343.925,Z 388.596,A -85,B 0,C 180,E1 -14145.706,E2 -14145.706} C_VEL
LIN {X 0,Y 344.581,Z 344.522,A -85,B 0,C 180,E1 -14146.744,E2 -14146.744} C_VEL
LIN {X 0,Y 340.973,Z 311.508,A -85,B 0,C 180,E1 -14147.699,E2 -14147.699} C_VEL
LIN {X 0,Y 342.004,Z 298.471,A -85,B 0,C 180,E1 -14151.076,E2 -14151.076} C_VEL
LIN {X 0,Y 343.067,Z 286.552,A -85,B 0,C 180,E1 -14154.187,E2 -14154.187} C_VEL
LIN {X 0,Y 342.002,Z 279.21,A -85,B 0,C 180,E1 -14156.22,E2 -14156.22} C_VEL
LIN {X 0,Y 340.815,Z 272.845,A -85,B 0,C 180,E1 -14158.055,E2 -14158.055} C_VEL
LIN {X 0,Y 340.699,Z 272.857,A -85,B 0,C 180,E1 -14161.044,E2 -14161.044} C_VEL
LIN {X 0,Y 340.719,Z 272.856,A -85,B 0,C 180,E1 -14165.278,E2 -14165.278} C_VEL
LIN {X 0,Y 340.712,Z 272.854,A -85,B 0,C 180,E1 -14168.386,E2 -14168.386} C_VEL
LIN {X 0,Y 340.699,Z 272.857,A -85,B 0,C 180,E1 -14172.045,E2 -14172.045} C_VEL
LIN {X 0,Y 340.652,Z 272.862,A -85,B 0,C 180,E1 -14176.226,E2 -14176.226} C_VEL
LIN {X 0,Y 340.688,Z 272.861,A -85,B 0,C 180,E1 -14179.752,E2 -14179.752} C_VEL
LIN {X 0,Y 340.704,Z 272.857,A -85,B 0,C 180,E1 -14183.257,E2 -14183.257} C_VEL
LIN {X 0,Y 340.693,Z 272.857,A -85,B 0,C 180,E1 -14186.153,E2 -14186.153} C_VEL
LIN {X 0,Y 340.773,Z 272.846,A -85,B 0,C 180,E1 -14190.331,E2 -14190.331} C_VEL
LIN {X 0,Y 340.803,Z 272.843,A -85,B 0,C 180,E1 -14193.019,E2 -14193.019} C_VEL
LIN {X 0,Y 340.726,Z 272.852,A -85,B 0,C 180,E1 -14196.926,E2 -14196.926} C_VEL
LIN {X 0,Y 340.789,Z 272.844,A -85,B 0,C 180,E1 -14200.733,E2 -14200.733} C_VEL
LIN {X 0,Y 340.783,Z 272.847,A -85,B 0,C 180,E1 -14203.218,E2 -14203.218} C_VEL
LIN {X 0,Y 340.841,Z 272.838,A -85,B 0,C 180,E1 -14206.889,E2 -14206.889} C_VEL
LIN {X 0,Y 340.91,Z 272.829,A -85,B 0,C 180,E1 -14210.506,E2 -14210.506} C_VEL
LIN {X 0,Y 341.055,Z 272.811,A -85,B 0,C 180,E1 -14212.897,E2 -14212.897} C_VEL
LIN {X 0,Y 341.165,Z 272.803,A -85,B 0,C 180,E1 -14217.638,E2 -14217.638} C_VEL
LIN {X 0,Y 341.291,Z 272.784,A -85,B 0,C 180,E1 -14219.999,E2 -14219.999} C_VEL
LIN {X 0,Y 341.165,Z 272.798,A -85,B 0,C 180,E1 -14222.36,E2 -14222.36} C_VEL
LIN {X 0,Y 341.07,Z 272.81,A -85,B 0,C 180,E1 -14227.101,E2 -14227.101} C_VEL
LIN {X 0,Y 340.869,Z 272.834,A -85,B 0,C 180,E1 -14230.693,E2 -14230.693} C_VEL
LIN {X 0,Y 340.857,Z 272.836,A -85,B 0,C 180,E1 -14234.324,E2 -14234.324} C_VEL
LIN {X 0,Y 340.832,Z 272.839,A -85,B 0,C 180,E1 -14238.466,E2 -14238.466} C_VEL
LIN {X 0,Y 340.747,Z 272.854,A -85,B 0,C 180,E1 -14241.856,E2 -14241.856} C_VEL
LIN {X 0,Y 340.765,Z 272.853,A -85,B 0,C 180,E1 -14245.664,E2 -14245.664} C_VEL
LIN {X 0,Y 340.721,Z 272.853,A -85,B 0,C 180,E1 -14248.32,E2 -14248.32} C_VEL
LIN {X 0,Y 340.695,Z 272.856,A -85,B 0,C 180,E1 -14251.043,E2 -14251.043} C_VEL
LIN {X 0,Y 340.711,Z 272.856,A -85,B 0,C 180,E1 -14255.278,E2 -14255.278} C_VEL
LIN {X 0,Y 340.711,Z 272.854,A -85,B 0,C 180,E1 -14258.387,E2 -14258.387} C_VEL
LIN {X 0,Y 340.726,Z 272.855,A -85,B 0,C 180,E1 -14262.051,E2 -14262.051} C_VEL
LIN {X 0,Y 340.727,Z 272.853,A -85,B 0,C 180,E1 -14266.212,E2 -14266.212} C_VEL
LIN {X 0,Y 340.756,Z 272.854,A -85,B 0,C 180,E1 -14269.737,E2 -14269.737} C_VEL
LIN {X 0,Y 340.702,Z 272.859,A -85,B 0,C 180,E1 -14273.559,E2 -14273.559} C_VEL
LIN {X 0,Y 340.684,Z 272.859,A -85,B 0,C 180,E1 -14276.153,E2 -14276.153} C_VEL
LIN {X 0,Y 340.766,Z 272.848,A -85,B 0,C 180,E1 -14280.332,E2 -14280.332} C_VEL
LIN {X 0,Y 340.796,Z 272.844,A -85,B 0,C 180,E1 -14283.02,E2 -14283.02} C_VEL
LIN {X 0,Y 340.721,Z 272.853,A -85,B 0,C 180,E1 -14286.927,E2 -14286.927} C_VEL
LIN {X 0,Y 340.787,Z 272.844,A -85,B 0,C 180,E1 -14290.733,E2 -14290.733} C_VEL
LIN {X 0,Y 340.778,Z 272.847,A -85,B 0,C 180,E1 -14293.218,E2 -14293.218} C_VEL
LIN {X 0,Y 340.836,Z 272.838,A -85,B 0,C 180,E1 -14296.89,E2 -14296.89} C_VEL
LIN {X 0,Y 340.92,Z 272.828,A -85,B 0,C 180,E1 -14300.507,E2 -14300.507} C_VEL
LIN {X 0,Y 341.066,Z 272.81,A -85,B 0,C 180,E1 -14302.898,E2 -14302.898} C_VEL
LIN {X 0,Y 341.158,Z 272.803,A -85,B 0,C 180,E1 -14307.638,E2 -14307.638} C_VEL
LIN {X 0,Y 341.287,Z 272.786,A -85,B 0,C 180,E1 -14310,E2 -14310} C_VEL
LIN {X 0,Y 341.159,Z 272.799,A -85,B 0,C 180,E1 -14312.361,E2 -14312.361} C_VEL
LIN {X 0,Y 341.051,Z 272.812,A -85,B 0,C 180,E1 -14317.102,E2 -14317.102} C_VEL
LIN {X 0,Y 340.866,Z 272.835,A -85,B 0,C 180,E1 -14320.693,E2 -14320.693} C_VEL
LIN {X 0,Y 340.854,Z 272.838,A -85,B 0,C 180,E1 -14324.325,E2 -14324.325} C_VEL
LIN {X 0,Y 340.827,Z 272.84,A -85,B 0,C 180,E1 -14328.466,E2 -14328.466} C_VEL
LIN {X 0,Y 340.712,Z 272.86,A -85,B 0,C 180,E1 -14331.843,E2 -14331.843} C_VEL
LIN {X 0,Y 340.761,Z 272.852,A -85,B 0,C 180,E1 -14335.664,E2 -14335.664} C_VEL
LIN {X 0,Y 340.727,Z 272.854,A -85,B 0,C 180,E1 -14338.32,E2 -14338.32} C_VEL
LIN {X 0,Y 340.778,Z 272.881,A -85,B 0,C 180,E1 -14340.743,E2 -14340.743} C_VEL
LIN {X 0,Y 341.201,Z 275.123,A -85,B 0,C 180,E1 -14341.424,E2 -14341.424} C_VEL
LIN {X 0,Y 343.61,Z 285.585,A -85,B 0,C 180,E1 -14341.78,E2 -14341.78} C_VEL
LIN {X 0,Y 345.141,Z 294.176,A -85,B 0,C 180,E1 -14342.049,E2 -14342.049} C_VEL
LIN {X 0,Y 344.159,Z 351.636,A -85,B 0,C 180,E1 -14343.395,E2 -14343.395} C_VEL
LIN {X 0,Y 343.845,Z 361.498,A -85,B 0,C 180,E1 -14343.78,E2 -14343.78} C_VEL
LIN {X 0,Y 343.46,Z 372.578,A -85,B 0,C 180,E1 -14344.42,E2 -14344.42} C_VEL
LIN {X 0,Y 342.927,Z 382.216,A -85,B 0,C 180,E1 -14345.196,E2 -14345.196} C_VEL
LIN {X 0,Y 342.443,Z 391.438,A -85,B 0,C 180,E1 -14346.159,E2 -14346.159} C_VEL
LIN {X 0,Y 341.918,Z 398.441,A -85,B 0,C 180,E1 -14347.048,E2 -14347.048} C_VEL
LIN {X 0,Y 341.31,Z 405.622,A -85,B 0,C 180,E1 -14348.15,E2 -14348.15} C_VEL
LIN {X 0,Y 340.917,Z 410.705,A -85,B 0,C 180,E1 -14349.074,E2 -14349.074} C_VEL
LIN {X 0,Y 340.467,Z 416.934,A -85,B 0,C 180,E1 -14350.443,E2 -14350.443} C_VEL
LIN {X 0,Y 340.11,Z 420.613,A -85,B 0,C 180,E1 -14351.393,E2 -14351.393} C_VEL
LIN {X 0,Y 339.902,Z 424.035,A -85,B 0,C 180,E1 -14352.434,E2 -14352.434} C_VEL
LIN {X 0,Y 339.579,Z 428.324,A -85,B 0,C 180,E1 -14354.12,E2 -14354.12} C_VEL
LIN {X 0,Y 338.809,Z 430.278,A -85,B 0,C 180,E1 -14355.052,E2 -14355.052} C_VEL
LIN {X 0,Y 337.102,Z 431.881,A -85,B 0,C 180,E1 -14355.979,E2 -14355.979} C_VEL
LIN {X 0,Y 333.181,Z 434.069,A -85,B 0,C 180,E1 -14357.876,E2 -14357.876} C_VEL
LIN {X 0,Y 332.094,Z 434.681,A -85,B 0,C 180,E1 -14358.878,E2 -14358.878} C_VEL
LIN {X 0,Y 332.01,Z 434.782,A -85,B 0,C 180,E1 -14359.219,E2 -14359.219} C_VEL
LIN {X 0,Y 332.218,Z 434.548,A -85,B 0,C 180,E1 -14361.509,E2 -14361.509} C_VEL
LIN {X 0,Y 332.643,Z 432.428,A -85,B 0,C 180,E1 -14363.733,E2 -14363.733} C_VEL
LIN {X 0,Y 333.076,Z 429.753,A -85,B 0,C 180,E1 -14365.375,E2 -14365.375} C_VEL
LIN {X 0,Y 333.579,Z 426.568,A -85,B 0,C 180,E1 -14366.787,E2 -14366.787} C_VEL
LIN {X 0,Y 334.313,Z 421.248,A -85,B 0,C 180,E1 -14368.593,E2 -14368.593} C_VEL
LIN {X 0,Y 335.087,Z 415.264,A -85,B 0,C 180,E1 -14370.126,E2 -14370.126} C_VEL
LIN {X 0,Y 335.989,Z 408.683,A -85,B 0,C 180,E1 -14371.463,E2 -14371.463} C_VEL
LIN {X 0,Y 336.877,Z 401.319,A -85,B 0,C 180,E1 -14372.681,E2 -14372.681} C_VEL
LIN {X 0,Y 337.714,Z 393.902,A -85,B 0,C 180,E1 -14373.684,E2 -14373.684} C_VEL
LIN {X 0,Y 338.333,Z 386.933,A -85,B 0,C 180,E1 -14374.469,E2 -14374.469} C_VEL
LIN {X 0,Y 339.127,Z 377.105,A -85,B 0,C 180,E1 -14375.352,E2 -14375.352} C_VEL
LIN {X 0,Y 339.889,Z 365.115,A -85,B 0,C 180,E1 -14376.142,E2 -14376.142} C_VEL
LIN {X 0,Y 340.261,Z 354.678,A -85,B 0,C 180,E1 -14376.593,E2 -14376.593} C_VEL
LIN {X 0,Y 341.152,Z 319.051,A -85,B 0,C 180,E1 -14377.491,E2 -14377.491} C_VEL
LIN {X 0,Y 341.727,Z 296.933,A -85,B 0,C 180,E1 -14378.029,E2 -14378.029} C_VEL
LIN {X 0,Y 340.455,Z 291.633,A -85,B 0,C 180,E1 -14378.265,E2 -14378.265} C_VEL
LIN {X 0,Y 334.284,Z 276.425,A -85,B 0,C 180,E1 -14379.181,E2 -14379.181} C_VEL
LIN {X 0,Y 333.724,Z 273.736,A -85,B 0,C 180,E1 -14380.07,E2 -14380.07} C_VEL
LIN {X 0,Y 333.737,Z 273.728,A -85,B 0,C 180,E1 -14382.855,E2 -14382.855} C_VEL
LIN {X 0,Y 333.787,Z 273.721,A -85,B 0,C 180,E1 -14386.609,E2 -14386.609} C_VEL
LIN {X 0,Y 333.842,Z 273.713,A -85,B 0,C 180,E1 -14390.305,E2 -14390.305} C_VEL
LIN {X 0,Y 334,Z 273.693,A -85,B 0,C 180,E1 -14392.748,E2 -14392.748} C_VEL
LIN {X 0,Y 333.805,Z 273.715,A -85,B 0,C 180,E1 -14395.17,E2 -14395.17} C_VEL
LIN {X 0,Y 334.1,Z 273.676,A -85,B 0,C 180,E1 -14397.59,E2 -14397.59} C_VEL
LIN {X 0,Y 334.239,Z 273.664,A -85,B 0,C 180,E1 -14400.001,E2 -14400.001} C_VEL
LIN {X 0,Y 334.1,Z 273.681,A -85,B 0,C 180,E1 -14402.412,E2 -14402.412} C_VEL
LIN {X 0,Y 334.018,Z 273.687,A -85,B 0,C 180,E1 -14407.254,E2 -14407.254} C_VEL
LIN {X 0,Y 333.826,Z 273.713,A -85,B 0,C 180,E1 -14410.923,E2 -14410.923} C_VEL
LIN {X 0,Y 333.802,Z 273.719,A -85,B 0,C 180,E1 -14414.635,E2 -14414.635} C_VEL
LIN {X 0,Y 333.791,Z 273.72,A -85,B 0,C 180,E1 -14418.656,E2 -14418.656} C_VEL
LIN {X 0,Y 333.687,Z 273.727,A -85,B 0,C 180,E1 -14422.279,E2 -14422.279} C_VEL
LIN {X 0,Y 333.731,Z 273.72,A -85,B 0,C 180,E1 -14426.247,E2 -14426.247} C_VEL
LIN {X 0,Y 333.707,Z 273.72,A -85,B 0,C 180,E1 -14428.973,E2 -14428.973} C_VEL
LIN {X 0,Y 333.639,Z 273.733,A -85,B 0,C 180,E1 -14432.588,E2 -14432.588} C_VEL
LIN {X 0,Y 333.673,Z 273.734,A -85,B 0,C 180,E1 -14436.14,E2 -14436.14} C_VEL
LIN {X 0,Y 333.669,Z 273.734,A -85,B 0,C 180,E1 -14439.19,E2 -14439.19} C_VEL
LIN {X 0,Y 333.672,Z 273.736,A -85,B 0,C 180,E1 -14442.509,E2 -14442.509} C_VEL
LIN {X 0,Y 333.618,Z 273.741,A -85,B 0,C 180,E1 -14445.96,E2 -14445.96} C_VEL
LIN {X 0,Y 333.646,Z 273.736,A -85,B 0,C 180,E1 -14449.317,E2 -14449.317} C_VEL
LIN {X 0,Y 333.666,Z 273.734,A -85,B 0,C 180,E1 -14453.169,E2 -14453.169} C_VEL
LIN {X 0,Y 333.636,Z 273.739,A -85,B 0,C 180,E1 -14456.793,E2 -14456.793} C_VEL
LIN {X 0,Y 333.739,Z 273.916,A -85,B 0,C 180,E1 -14460.6,E2 -14460.6} C_VEL
LIN {X 0,Y 335.755,Z 282.901,A -85,B 0,C 180,E1 -14463.255,E2 -14463.255} C_VEL
LIN {X 0,Y 336.869,Z 290.346,A -85,B 0,C 180,E1 -14465.339,E2 -14465.339} C_VEL
LIN {X 0,Y 335.305,Z 306.497,A -85,B 0,C 180,E1 -14469.447,E2 -14469.447} C_VEL
LIN {X 0,Y 335.156,Z 308.42,A -85,B 0,C 180,E1 -14469.933,E2 -14469.933} C_VEL
LIN {X 0,Y 338.931,Z 330.042,A -85,B 0,C 180,E1 -14470.814,E2 -14470.814} C_VEL
LIN {X 0,Y 340.743,Z 346.861,A -85,B 0,C 180,E1 -14471.384,E2 -14471.384} C_VEL
LIN {X 0,Y 339.688,Z 388.314,A -85,B 0,C 180,E1 -14472.412,E2 -14472.412} C_VEL
LIN {X 0,Y 339.076,Z 399.824,A -85,B 0,C 180,E1 -14472.892,E2 -14472.892} C_VEL
LIN {X 0,Y 338.204,Z 410.28,A -85,B 0,C 180,E1 -14473.553,E2 -14473.553} C_VEL
LIN {X 0,Y 337.346,Z 419.042,A -85,B 0,C 180,E1 -14474.287,E2 -14474.287} C_VEL
LIN {X 0,Y 336.356,Z 427.458,A -85,B 0,C 180,E1 -14475.17,E2 -14475.17} C_VEL
LIN {X 0,Y 335.399,Z 435.456,A -85,B 0,C 180,E1 -14476.211,E2 -14476.211} C_VEL
LIN {X 0,Y 334.585,Z 442.095,A -85,B 0,C 180,E1 -14477.259,E2 -14477.259} C_VEL
LIN {X 0,Y 333.881,Z 448.436,A -85,B 0,C 180,E1 -14478.465,E2 -14478.465} C_VEL
LIN {X 0,Y 333.21,Z 453.722,A -85,B 0,C 180,E1 -14479.673,E2 -14479.673} C_VEL
LIN {X 0,Y 332.75,Z 458.141,A -85,B 0,C 180,E1 -14480.886,E2 -14480.886} C_VEL
LIN {X 0,Y 332.442,Z 461.826,A -85,B 0,C 180,E1 -14482.102,E2 -14482.102} C_VEL
LIN {X 0,Y 332.103,Z 466.079,A -85,B 0,C 180,E1 -14483.927,E2 -14483.927} C_VEL
LIN {X 0,Y 332.054,Z 468.192,A -85,B 0,C 180,E1 -14485.144,E2 -14485.144} C_VEL
LIN {X 0,Y 332.063,Z 469.785,A -85,B 0,C 180,E1 -14486.36,E2 -14486.36} C_VEL
LIN {X 0,Y 332.043,Z 470.835,A -85,B 0,C 180,E1 -14487.574,E2 -14487.574} C_VEL
LIN {X 0,Y 332.154,Z 471.286,A -85,B 0,C 180,E1 -14488.788,E2 -14488.788} C_VEL
LIN {X 0,Y 332.265,Z 471.239,A -85,B 0,C 180,E1 -14490,E2 -14490} C_VEL
LIN {X 0,Y 332.2,Z 470.695,A -85,B 0,C 180,E1 -14491.213,E2 -14491.213} C_VEL
LIN {X 0,Y 332.093,Z 469.649,A -85,B 0,C 180,E1 -14492.426,E2 -14492.426} C_VEL
LIN {X 0,Y 332.156,Z 466.93,A -85,B 0,C 180,E1 -14494.247,E2 -14494.247} C_VEL
LIN {X 0,Y 332.151,Z 462.894,A -85,B 0,C 180,E1 -14496.073,E2 -14496.073} C_VEL
LIN {X 0,Y 332.312,Z 459.372,A -85,B 0,C 180,E1 -14497.29,E2 -14497.29} C_VEL
LIN {X 0,Y 332.609,Z 453.903,A -85,B 0,C 180,E1 -14498.812,E2 -14498.812} C_VEL
LIN {X 0,Y 333.073,Z 447.062,A -85,B 0,C 180,E1 -14500.332,E2 -14500.332} C_VEL
LIN {X 0,Y 333.722,Z 438.233,A -85,B 0,C 180,E1 -14501.849,E2 -14501.849} C_VEL
LIN {X 0,Y 334.415,Z 430.55,A -85,B 0,C 180,E1 -14502.903,E2 -14502.903} C_VEL
LIN {X 0,Y 335.037,Z 422.495,A -85,B 0,C 180,E1 -14503.805,E2 -14503.805} C_VEL
LIN {X 0,Y 335.547,Z 414.179,A -85,B 0,C 180,E1 -14504.557,E2 -14504.557} C_VEL
LIN {X 0,Y 336.198,Z 404.612,A -85,B 0,C 180,E1 -14505.225,E2 -14505.225} C_VEL
LIN {X 0,Y 336.853,Z 392.76,A -85,B 0,C 180,E1 -14505.81,E2 -14505.81} C_VEL
LIN {X 0,Y 337.224,Z 375.232,A -85,B 0,C 180,E1 -14506.28,E2 -14506.28} C_VEL
LIN {X 0,Y 337.599,Z 344.479,A -85,B 0,C 180,E1 -14507.008,E2 -14507.008} C_VEL
LIN {X 0,Y 333.98,Z 311.113,A -85,B 0,C 180,E1 -14508.003,E2 -14508.003} C_VEL
LIN {X 0,Y 335.214,Z 296.614,A -85,B 0,C 180,E1 -14511.848,E2 -14511.848} C_VEL
LIN {X 0,Y 336.042,Z 287.068,A -85,B 0,C 180,E1 -14514.396,E2 -14514.396} C_VEL
LIN {X 0,Y 334.658,Z 278.459,A -85,B 0,C 180,E1 -14516.84,E2 -14516.84} C_VEL
LIN {X 0,Y 333.757,Z 273.724,A -85,B 0,C 180,E1 -14518.249,E2 -14518.249} C_VEL
LIN {X 0,Y 333.633,Z 273.739,A -85,B 0,C 180,E1 -14521.777,E2 -14521.777} C_VEL
LIN {X 0,Y 333.687,Z 273.729,A -85,B 0,C 180,E1 -14524.773,E2 -14524.773} C_VEL
LIN {X 0,Y 333.655,Z 273.738,A -85,B 0,C 180,E1 -14527.65,E2 -14527.65} C_VEL
LIN {X 0,Y 333.647,Z 273.734,A -85,B 0,C 180,E1 -14530.767,E2 -14530.767} C_VEL
LIN {X 0,Y 333.593,Z 273.741,A -85,B 0,C 180,E1 -14534.249,E2 -14534.249} C_VEL
LIN {X 0,Y 333.641,Z 273.74,A -85,B 0,C 180,E1 -14537.618,E2 -14537.618} C_VEL
LIN {X 0,Y 333.652,Z 273.735,A -85,B 0,C 180,E1 -14541.201,E2 -14541.201} C_VEL
LIN {X 0,Y 333.675,Z 273.733,A -85,B 0,C 180,E1 -14543.86,E2 -14543.86} C_VEL
LIN {X 0,Y 333.645,Z 273.738,A -85,B 0,C 180,E1 -14547.411,E2 -14547.411} C_VEL
LIN {X 0,Y 333.709,Z 273.727,A -85,B 0,C 180,E1 -14551.027,E2 -14551.027} C_VEL
LIN {X 0,Y 333.734,Z 273.727,A -85,B 0,C 180,E1 -14553.753,E2 -14553.753} C_VEL
LIN {X 0,Y 333.718,Z 273.728,A -85,B 0,C 180,E1 -14557.913,E2 -14557.913} C_VEL
LIN {X 0,Y 333.791,Z 273.722,A -85,B 0,C 180,E1 -14561.588,E2 -14561.588} C_VEL
LIN {X 0,Y 333.805,Z 273.72,A -85,B 0,C 180,E1 -14565.576,E2 -14565.576} C_VEL
LIN {X 0,Y 333.83,Z 273.712,A -85,B 0,C 180,E1 -14569.077,E2 -14569.077} C_VEL
LIN {X 0,Y 334.002,Z 273.689,A -85,B 0,C 180,E1 -14572.746,E2 -14572.746} C_VEL
LIN {X 0,Y 333.806,Z 273.716,A -85,B 0,C 180,E1 -14575.168,E2 -14575.168} C_VEL
LIN {X 0,Y 334.102,Z 273.683,A -85,B 0,C 180,E1 -14577.588,E2 -14577.588} C_VEL
LIN {X 0,Y 334.242,Z 273.662,A -85,B 0,C 180,E1 -14579.999,E2 -14579.999} C_VEL
LIN {X 0,Y 334.102,Z 273.677,A -85,B 0,C 180,E1 -14582.41,E2 -14582.41} C_VEL
LIN {X 0,Y 334.02,Z 273.689,A -85,B 0,C 180,E1 -14587.251,E2 -14587.251} C_VEL
LIN {X 0,Y 333.831,Z 273.711,A -85,B 0,C 180,E1 -14590.921,E2 -14590.921} C_VEL
LIN {X 0,Y 333.803,Z 273.714,A -85,B 0,C 180,E1 -14594.633,E2 -14594.633} C_VEL
LIN {X 0,Y 333.791,Z 273.716,A -85,B 0,C 180,E1 -14598.655,E2 -14598.655} C_VEL
LIN {X 0,Y 333.686,Z 273.73,A -85,B 0,C 180,E1 -14602.277,E2 -14602.277} C_VEL
LIN {X 0,Y 333.728,Z 273.725,A -85,B 0,C 180,E1 -14606.246,E2 -14606.246} C_VEL
LIN {X 0,Y 333.697,Z 273.728,A -85,B 0,C 180,E1 -14610.289,E2 -14610.289} C_VEL
LIN {X 0,Y 333.666,Z 273.731,A -85,B 0,C 180,E1 -14614.658,E2 -14614.658} C_VEL
LIN {X 0,Y 333.65,Z 273.739,A -85,B 0,C 180,E1 -14617.65,E2 -14617.65} C_VEL
LIN {X 0,Y 333.648,Z 273.734,A -85,B 0,C 180,E1 -14620.765,E2 -14620.765} C_VEL
LIN {X 0,Y 333.655,Z 273.734,A -85,B 0,C 180,E1 -14624.262,E2 -14624.262} C_VEL
LIN {X 0,Y 333.688,Z 273.734,A -85,B 0,C 180,E1 -14627.626,E2 -14627.626} C_VEL
LIN {X 0,Y 333.674,Z 273.732,A -85,B 0,C 180,E1 -14631.195,E2 -14631.195} C_VEL
LIN {X 0,Y 333.677,Z 273.731,A -85,B 0,C 180,E1 -14635.225,E2 -14635.225} C_VEL
LIN {X 0,Y 333.689,Z 273.733,A -85,B 0,C 180,E1 -14639.637,E2 -14639.637} C_VEL
LIN {X 0,Y 333.735,Z 273.724,A -85,B 0,C 180,E1 -14642.401,E2 -14642.401} C_VEL
LIN {X 0,Y 333.718,Z 273.725,A -85,B 0,C 180,E1 -14645.09,E2 -14645.09} C_VEL
LIN {X 0,Y 333.674,Z 273.731,A -85,B 0,C 180,E1 -14649.019,E2 -14649.019} C_VEL
LIN {X 0,Y 333.786,Z 273.72,A -85,B 0,C 180,E1 -14651.589,E2 -14651.589} C_VEL
LIN {X 0,Y 333.8,Z 273.719,A -85,B 0,C 180,E1 -14655.576,E2 -14655.576} C_VEL
LIN {X 0,Y 333.826,Z 273.712,A -85,B 0,C 180,E1 -14659.078,E2 -14659.078} C_VEL
LIN {X 0,Y 334.016,Z 273.688,A -85,B 0,C 180,E1 -14662.747,E2 -14662.747} C_VEL
LIN {X 0,Y 333.799,Z 273.716,A -85,B 0,C 180,E1 -14665.169,E2 -14665.169} C_VEL
LIN {X 0,Y 334.096,Z 273.682,A -85,B 0,C 180,E1 -14667.589,E2 -14667.589} C_VEL
LIN {X 0,Y 334.238,Z 273.664,A -85,B 0,C 180,E1 -14670,E2 -14670} C_VEL
LIN {X 0,Y 334.096,Z 273.679,A -85,B 0,C 180,E1 -14672.411,E2 -14672.411} C_VEL
LIN {X 0,Y 334.005,Z 273.693,A -85,B 0,C 180,E1 -14676.039,E2 -14676.039} C_VEL
LIN {X 0,Y 333.976,Z 273.693,A -85,B 0,C 180,E1 -14678.501,E2 -14678.501} C_VEL
LIN {X 0,Y 333.786,Z 273.719,A -85,B 0,C 180,E1 -14682.154,E2 -14682.154} C_VEL
LIN {X 0,Y 333.768,Z 273.724,A -85,B 0,C 180,E1 -14685.886,E2 -14685.886} C_VEL
LIN {X 0,Y 333.786,Z 273.717,A -85,B 0,C 180,E1 -14688.654,E2 -14688.654} C_VEL
LIN {X 0,Y 333.65,Z 273.735,A -85,B 0,C 180,E1 -14692.28,E2 -14692.28} C_VEL
LIN {X 0,Y 333.724,Z 273.726,A -85,B 0,C 180,E1 -14696.246,E2 -14696.246} C_VEL
LIN {X 0,Y 333.713,Z 273.729,A -85,B 0,C 180,E1 -14700.36,E2 -14700.36} C_VEL
LIN {X 0,Y 333.746,Z 273.832,A -85,B 0,C 180,E1 -14700.619,E2 -14700.619} C_VEL
LIN {X 0,Y 334.04,Z 275.43,A -85,B 0,C 180,E1 -14701.115,E2 -14701.115} C_VEL
LIN {X 0,Y 336.528,Z 285.402,A -85,B 0,C 180,E1 -14701.472,E2 -14701.472} C_VEL
LIN {X 0,Y 338.283,Z 296.322,A -85,B 0,C 180,E1 -14701.814,E2 -14701.814} C_VEL
LIN {X 0,Y 337.195,Z 352.97,A -85,B 0,C 180,E1 -14703.177,E2 -14703.177} C_VEL
LIN {X 0,Y 336.891,Z 364.05,A -85,B 0,C 180,E1 -14703.645,E2 -14703.645} C_VEL
LIN {X 0,Y 336.305,Z 376.004,A -85,B 0,C 180,E1 -14704.432,E2 -14704.432} C_VEL
LIN {X 0,Y 335.836,Z 384.712,A -85,B 0,C 180,E1 -14705.198,E2 -14705.198} C_VEL
LIN {X 0,Y 335.388,Z 392.983,A -85,B 0,C 180,E1 -14706.11,E2 -14706.11} C_VEL
LIN {X 0,Y 334.791,Z 400.308,A -85,B 0,C 180,E1 -14707.091,E2 -14707.091} C_VEL
LIN {X 0,Y 334.1,Z 408.049,A -85,B 0,C 180,E1 -14708.355,E2 -14708.355} C_VEL
LIN {X 0,Y 333.541,Z 415.561,A -85,B 0,C 180,E1 -14709.896,E2 -14709.896} C_VEL
LIN {X 0,Y 332.966,Z 421.931,A -85,B 0,C 180,E1 -14711.596,E2 -14711.596} C_VEL
LIN {X 0,Y 332.704,Z 425.825,A -85,B 0,C 180,E1 -14712.898,E2 -14712.898} C_VEL
LIN {X 0,Y 332.478,Z 429.014,A -85,B 0,C 180,E1 -14714.23,E2 -14714.23} C_VEL
LIN {X 0,Y 332.135,Z 432.109,A -85,B 0,C 180,E1 -14716.007,E2 -14716.007} C_VEL
LIN {X 0,Y 331.996,Z 434.068,A -85,B 0,C 180,E1 -14717.808,E2 -14717.808} C_VEL
LIN {X 0,Y 332.01,Z 434.782,A -85,B 0,C 180,E1 -14719.219,E2 -14719.219} C_VEL
LIN {X 0,Y 331.389,Z 434.995,A -85,B 0,C 180,E1 -14720.235,E2 -14720.235} C_VEL
LIN {X 0,Y 328.728,Z 434.654,A -85,B 0,C 180,E1 -14721.895,E2 -14721.895} C_VEL
LIN {X 0,Y 326.187,Z 433.324,A -85,B 0,C 180,E1 -14723.562,E2 -14723.562} C_VEL
LIN {X 0,Y 325.765,Z 431.943,A -85,B 0,C 180,E1 -14724.573,E2 -14724.573} C_VEL
LIN {X 0,Y 326.428,Z 428.17,A -85,B 0,C 180,E1 -14726.549,E2 -14726.549} C_VEL
LIN {X 0,Y 326.913,Z 424.824,A -85,B 0,C 180,E1 -14727.856,E2 -14727.856} C_VEL
LIN {X 0,Y 327.704,Z 419.473,A -85,B 0,C 180,E1 -14729.478,E2 -14729.478} C_VEL
LIN {X 0,Y 328.519,Z 413.507,A -85,B 0,C 180,E1 -14730.92,E2 -14730.92} C_VEL
LIN {X 0,Y 329.604,Z 406.06,A -85,B 0,C 180,E1 -14732.362,E2 -14732.362} C_VEL
LIN {X 0,Y 330.693,Z 397.604,A -85,B 0,C 180,E1 -14733.665,E2 -14733.665} C_VEL
LIN {X 0,Y 331.585,Z 388.601,A -85,B 0,C 180,E1 -14734.752,E2 -14734.752} C_VEL
LIN {X 0,Y 332.317,Z 379.753,A -85,B 0,C 180,E1 -14735.602,E2 -14735.602} C_VEL
LIN {X 0,Y 333.017,Z 371.332,A -85,B 0,C 180,E1 -14736.228,E2 -14736.228} C_VEL
LIN {X 0,Y 333.437,Z 361.979,A -85,B 0,C 180,E1 -14736.764,E2 -14736.764} C_VEL
LIN {X 0,Y 333.772,Z 351.838,A -85,B 0,C 180,E1 -14737.158,E2 -14737.158} C_VEL
LIN {X 0,Y 335.172,Z 297.671,A -85,B 0,C 180,E1 -14738.514,E2 -14738.514} C_VEL
LIN {X 0,Y 333.668,Z 292.431,A -85,B 0,C 180,E1 -14738.777,E2 -14738.777} C_VEL
LIN {X 0,Y 328.041,Z 279.1,A -85,B 0,C 180,E1 -14739.628,E2 -14739.628} C_VEL
LIN {X 0,Y 327.18,Z 276.778,A -85,B 0,C 180,E1 -14739.818,E2 -14739.818} C_VEL
LIN {X 0,Y 326.724,Z 274.607,A -85,B 0,C 180,E1 -14740.526,E2 -14740.526} C_VEL
LIN {X 0,Y 326.719,Z 274.602,A -85,B 0,C 180,E1 -14743.762,E2 -14743.762} C_VEL
LIN {X 0,Y 326.75,Z 274.596,A -85,B 0,C 180,E1 -14746.315,E2 -14746.315} C_VEL
LIN {X 0,Y 326.797,Z 274.59,A -85,B 0,C 180,E1 -14750.094,E2 -14750.094} C_VEL
LIN {X 0,Y 326.984,Z 274.568,A -85,B 0,C 180,E1 -14753.832,E2 -14753.832} C_VEL
LIN {X 0,Y 327.04,Z 274.555,A -85,B 0,C 180,E1 -14757.538,E2 -14757.538} C_VEL
LIN {X 0,Y 327.19,Z 274.542,A -85,B 0,C 180,E1 -14760.001,E2 -14760.001} C_VEL
LIN {X 0,Y 327.04,Z 274.561,A -85,B 0,C 180,E1 -14762.464,E2 -14762.464} C_VEL
LIN {X 0,Y 326.989,Z 274.566,A -85,B 0,C 180,E1 -14766.17,E2 -14766.17} C_VEL
LIN {X 0,Y 326.908,Z 274.57,A -85,B 0,C 180,E1 -14768.656,E2 -14768.656} C_VEL
LIN {X 0,Y 326.727,Z 274.591,A -85,B 0,C 180,E1 -14772.423,E2 -14772.423} C_VEL
LIN {X 0,Y 326.748,Z 274.595,A -85,B 0,C 180,E1 -14774.959,E2 -14774.959} C_VEL
LIN {X 0,Y 326.727,Z 274.598,A -85,B 0,C 180,E1 -14778.839,E2 -14778.839} C_VEL
LIN {X 0,Y 326.616,Z 274.613,A -85,B 0,C 180,E1 -14782.789,E2 -14782.789} C_VEL
LIN {X 0,Y 326.685,Z 274.594,A -85,B 0,C 180,E1 -14785.485,E2 -14785.485} C_VEL
LIN {X 0,Y 326.657,Z 274.597,A -85,B 0,C 180,E1 -14789.66,E2 -14789.66} C_VEL
LIN {X 0,Y 326.603,Z 274.606,A -85,B 0,C 180,E1 -14794.021,E2 -14794.021} C_VEL
LIN {X 0,Y 326.626,Z 274.604,A -85,B 0,C 180,E1 -14797.24,E2 -14797.24} C_VEL
LIN {X 0,Y 326.601,Z 274.612,A -85,B 0,C 180,E1 -14800.208,E2 -14800.208} C_VEL
LIN {X 0,Y 326.599,Z 274.611,A -85,B 0,C 180,E1 -14803.52,E2 -14803.52} C_VEL
LIN {X 0,Y 326.58,Z 274.616,A -85,B 0,C 180,E1 -14807.028,E2 -14807.028} C_VEL
LIN {X 0,Y 326.611,Z 274.614,A -85,B 0,C 180,E1 -14810.774,E2 -14810.774} C_VEL
LIN {X 0,Y 326.613,Z 274.616,A -85,B 0,C 180,E1 -14814.482,E2 -14814.482} C_VEL
LIN {X 0,Y 326.607,Z 274.615,A -85,B 0,C 180,E1 -14817.457,E2 -14817.457} C_VEL
LIN {X 0,Y 326.69,Z 274.792,A -85,B 0,C 180,E1 -14820.116,E2 -14820.116} C_VEL
LIN {X 0,Y 328.829,Z 284.197,A -85,B 0,C 180,E1 -14822.989,E2 -14822.989} C_VEL
LIN {X 0,Y 329.901,Z 290.393,A -85,B 0,C 180,E1 -14824.783,E2 -14824.783} C_VEL
LIN {X 0,Y 329.599,Z 295.354,A -85,B 0,C 180,E1 -14826.101,E2 -14826.101} C_VEL
LIN {X 0,Y 328.366,Z 308.308,A -85,B 0,C 180,E1 -14829.399,E2 -14829.399} C_VEL
LIN {X 0,Y 332.062,Z 328.747,A -85,B 0,C 180,E1 -14830.26,E2 -14830.26} C_VEL
LIN {X 0,Y 334.126,Z 345.968,A -85,B 0,C 180,E1 -14830.877,E2 -14830.877} C_VEL
LIN {X 0,Y 333.138,Z 387.475,A -85,B 0,C 180,E1 -14831.94,E2 -14831.94} C_VEL
LIN {X 0,Y 332.527,Z 398.724,A -85,B 0,C 180,E1 -14832.411,E2 -14832.411} C_VEL
LIN {X 0,Y 331.614,Z 409.1,A -85,B 0,C 180,E1 -14833.058,E2 -14833.058} C_VEL
LIN {X 0,Y 330.543,Z 419.476,A -85,B 0,C 180,E1 -14833.955,E2 -14833.955} C_VEL
LIN {X 0,Y 329.525,Z 427.72,A -85,B 0,C 180,E1 -14834.856,E2 -14834.856} C_VEL
LIN {X 0,Y 328.528,Z 435.603,A -85,B 0,C 180,E1 -14835.917,E2 -14835.917} C_VEL
LIN {X 0,Y 327.673,Z 442.156,A -85,B 0,C 180,E1 -14836.986,E2 -14836.986} C_VEL
LIN {X 0,Y 326.933,Z 448.423,A -85,B 0,C 180,E1 -14838.217,E2 -14838.217} C_VEL
LIN {X 0,Y 326.058,Z 454.853,A -85,B 0,C 180,E1 -14839.757,E2 -14839.757} C_VEL
LIN {X 0,Y 325.534,Z 459.983,A -85,B 0,C 180,E1 -14841.308,E2 -14841.308} C_VEL
LIN {X 0,Y 325.144,Z 464.626,A -85,B 0,C 180,E1 -14843.173,E2 -14843.173} C_VEL
LIN {X 0,Y 324.961,Z 467.904,A -85,B 0,C 180,E1 -14845.038,E2 -14845.038} C_VEL
LIN {X 0,Y 324.987,Z 469.452,A -85,B 0,C 180,E1 -14846.281,E2 -14846.281} C_VEL
LIN {X 0,Y 324.955,Z 470.48,A -85,B 0,C 180,E1 -14847.521,E2 -14847.521} C_VEL
LIN {X 0,Y 325.057,Z 470.908,A -85,B 0,C 180,E1 -14848.761,E2 -14848.761} C_VEL
LIN {X 0,Y 325.187,Z 470.82,A -85,B 0,C 180,E1 -14850,E2 -14850} C_VEL
LIN {X 0,Y 325.107,Z 470.234,A -85,B 0,C 180,E1 -14851.239,E2 -14851.239} C_VEL
LIN {X 0,Y 325.003,Z 469.145,A -85,B 0,C 180,E1 -14852.479,E2 -14852.479} C_VEL
LIN {X 0,Y 325.085,Z 466.382,A -85,B 0,C 180,E1 -14854.34,E2 -14854.34} C_VEL
LIN {X 0,Y 325.072,Z 462.804,A -85,B 0,C 180,E1 -14856.001,E2 -14856.001} C_VEL
LIN {X 0,Y 325.263,Z 458.717,A -85,B 0,C 180,E1 -14857.449,E2 -14857.449} C_VEL
LIN {X 0,Y 325.566,Z 453.184,A -85,B 0,C 180,E1 -14859.004,E2 -14859.004} C_VEL
LIN {X 0,Y 326.051,Z 446.259,A -85,B 0,C 180,E1 -14860.557,E2 -14860.557} C_VEL
LIN {X 0,Y 326.776,Z 437.274,A -85,B 0,C 180,E1 -14862.104,E2 -14862.104} C_VEL
LIN {X 0,Y 327.478,Z 429.471,A -85,B 0,C 180,E1 -14863.181,E2 -14863.181} C_VEL
LIN {X 0,Y 328.137,Z 421.27,A -85,B 0,C 180,E1 -14864.101,E2 -14864.101} C_VEL
LIN {X 0,Y 328.626,Z 412.745,A -85,B 0,C 180,E1 -14864.87,E2 -14864.87} C_VEL
LIN {X 0,Y 329.414,Z 401.685,A -85,B 0,C 180,E1 -14865.626,E2 -14865.626} C_VEL
LIN {X 0,Y 329.933,Z 390.728,A -85,B 0,C 180,E1 -14866.119,E2 -14866.119} C_VEL
LIN {X 0,Y 330.398,Z 367.419,A -85,B 0,C 180,E1 -14866.725,E2 -14866.725} C_VEL
LIN {X 0,Y 330.701,Z 345.228,A -85,B 0,C 180,E1 -14867.263,E2 -14867.263} C_VEL
LIN {X 0,Y 326.982,Z 310.726,A -85,B 0,C 180,E1 -14868.321,E2 -14868.321} C_VEL
LIN {X 0,Y 328.196,Z 297.102,A -85,B 0,C 180,E1 -14872.008,E2 -14872.008} C_VEL
LIN {X 0,Y 329.005,Z 288.757,A -85,B 0,C 180,E1 -14874.28,E2 -14874.28} C_VEL
LIN {X 0,Y 328.091,Z 281.834,A -85,B 0,C 180,E1 -14876.274,E2 -14876.274} C_VEL
LIN {X 0,Y 326.711,Z 274.601,A -85,B 0,C 180,E1 -14878.42,E2 -14878.42} C_VEL
LIN {X 0,Y 326.609,Z 274.61,A -85,B 0,C 180,E1 -14882.544,E2 -14882.544} C_VEL
LIN {X 0,Y 326.615,Z 274.615,A -85,B 0,C 180,E1 -14885.519,E2 -14885.519} C_VEL
LIN {X 0,Y 326.613,Z 274.613,A -85,B 0,C 180,E1 -14889.226,E2 -14889.226} C_VEL
LIN {X 0,Y 326.576,Z 274.615,A -85,B 0,C 180,E1 -14892.971,E2 -14892.971} C_VEL
LIN {X 0,Y 326.576,Z 274.616,A -85,B 0,C 180,E1 -14897.027,E2 -14897.027} C_VEL
LIN {X 0,Y 326.611,Z 274.61,A -85,B 0,C 180,E1 -14900.772,E2 -14900.772} C_VEL
LIN {X 0,Y 326.611,Z 274.61,A -85,B 0,C 180,E1 -14904.479,E2 -14904.479} C_VEL
LIN {X 0,Y 326.609,Z 274.615,A -85,B 0,C 180,E1 -14907.455,E2 -14907.455} C_VEL
LIN {X 0,Y 326.659,Z 274.604,A -85,B 0,C 180,E1 -14910.34,E2 -14910.34} C_VEL
LIN {X 0,Y 326.688,Z 274.6,A -85,B 0,C 180,E1 -14914.515,E2 -14914.515} C_VEL
LIN {X 0,Y 326.644,Z 274.606,A -85,B 0,C 180,E1 -14918.544,E2 -14918.544} C_VEL
LIN {X 0,Y 326.742,Z 274.596,A -85,B 0,C 180,E1 -14921.176,E2 -14921.176} C_VEL
LIN {X 0,Y 326.76,Z 274.596,A -85,B 0,C 180,E1 -14925.432,E2 -14925.432} C_VEL
LIN {X 0,Y 326.766,Z 274.591,A -85,B 0,C 180,E1 -14928.838,E2 -14928.838} C_VEL
LIN {X 0,Y 326.955,Z 274.567,A -85,B 0,C 180,E1 -14932.589,E2 -14932.589} C_VEL
LIN {X 0,Y 326.773,Z 274.591,A -85,B 0,C 180,E1 -14935.064,E2 -14935.064} C_VEL
LIN {X 0,Y 327.043,Z 274.561,A -85,B 0,C 180,E1 -14937.536,E2 -14937.536} C_VEL
LIN {X 0,Y 327.193,Z 274.54,A -85,B 0,C 180,E1 -14939.999,E2 -14939.999} C_VEL
LIN {X 0,Y 327.043,Z 274.556,A -85,B 0,C 180,E1 -14942.462,E2 -14942.462} C_VEL
LIN {X 0,Y 326.965,Z 274.566,A -85,B 0,C 180,E1 -14946.679,E2 -14946.679} C_VEL
LIN {X 0,Y 326.81,Z 274.589,A -85,B 0,C 180,E1 -14949.905,E2 -14949.905} C_VEL
LIN {X 0,Y 326.754,Z 274.598,A -85,B 0,C 180,E1 -14953.684,E2 -14953.684} C_VEL
LIN {X 0,Y 326.694,Z 274.604,A -85,B 0,C 180,E1 -14957.527,E2 -14957.527} C_VEL
LIN {X 0,Y 326.667,Z 274.605,A -85,B 0,C 180,E1 -14960.133,E2 -14960.133} C_VEL
LIN {X 0,Y 326.646,Z 274.608,A -85,B 0,C 180,E1 -14964.128,E2 -14964.128} C_VEL
LIN {X 0,Y 326.676,Z 274.602,A -85,B 0,C 180,E1 -14966.857,E2 -14966.857} C_VEL
LIN {X 0,Y 326.632,Z 274.607,A -85,B 0,C 180,E1 -14970.61,E2 -14970.61} C_VEL
LIN {X 0,Y 326.599,Z 274.614,A -85,B 0,C 180,E1 -14974.019,E2 -14974.019} C_VEL
LIN {X 0,Y 326.623,Z 274.61,A -85,B 0,C 180,E1 -14977.238,E2 -14977.238} C_VEL
LIN {X 0,Y 326.596,Z 274.613,A -85,B 0,C 180,E1 -14980.206,E2 -14980.206} C_VEL
LIN {X 0,Y 326.602,Z 274.615,A -85,B 0,C 180,E1 -14983.517,E2 -14983.517} C_VEL
LIN {X 0,Y 326.625,Z 274.609,A -85,B 0,C 180,E1 -14987.017,E2 -14987.017} C_VEL
LIN {X 0,Y 326.637,Z 274.607,A -85,B 0,C 180,E1 -14990.765,E2 -14990.765} C_VEL
LIN {X 0,Y 326.604,Z 274.611,A -85,B 0,C 180,E1 -14994.48,E2 -14994.48} C_VEL
LIN {X 0,Y 326.599,Z 274.615,A -85,B 0,C 180,E1 -14997.455,E2 -14997.455} C_VEL
LIN {X 0,Y 326.652,Z 274.606,A -85,B 0,C 180,E1 -15000.34,E2 -15000.34} C_VEL
LIN {X 0,Y 326.682,Z 274.602,A -85,B 0,C 180,E1 -15004.516,E2 -15004.516} C_VEL
LIN {X 0,Y 326.639,Z 274.607,A -85,B 0,C 180,E1 -15008.545,E2 -15008.545} C_VEL
LIN {X 0,Y 326.736,Z 274.595,A -85,B 0,C 180,E1 -15011.177,E2 -15011.177} C_VEL
LIN {X 0,Y 326.755,Z 274.595,A -85,B 0,C 180,E1 -15015.433,E2 -15015.433} C_VEL
LIN {X 0,Y 326.762,Z 274.591,A -85,B 0,C 180,E1 -15018.839,E2 -15018.839} C_VEL
LIN {X 0,Y 326.97,Z 274.566,A -85,B 0,C 180,E1 -15022.59,E2 -15022.59} C_VEL
LIN {X 0,Y 326.766,Z 274.591,A -85,B 0,C 180,E1 -15025.064,E2 -15025.064} C_VEL
LIN {X 0,Y 327.036,Z 274.56,A -85,B 0,C 180,E1 -15027.536,E2 -15027.536} C_VEL
LIN {X 0,Y 327.19,Z 274.542,A -85,B 0,C 180,E1 -15030,E2 -15030} C_VEL
LIN {X 0,Y 327.037,Z 274.558,A -85,B 0,C 180,E1 -15032.463,E2 -15032.463} C_VEL
LIN {X 0,Y 326.98,Z 274.567,A -85,B 0,C 180,E1 -15036.169,E2 -15036.169} C_VEL
LIN {X 0,Y 326.906,Z 274.573,A -85,B 0,C 180,E1 -15038.655,E2 -15038.655} C_VEL
LIN {X 0,Y 326.729,Z 274.596,A -85,B 0,C 180,E1 -15042.421,E2 -15042.421} C_VEL
LIN {X 0,Y 326.745,Z 274.593,A -85,B 0,C 180,E1 -15044.957,E2 -15044.957} C_VEL
LIN {X 0,Y 326.723,Z 274.596,A -85,B 0,C 180,E1 -15048.838,E2 -15048.838} C_VEL
LIN {X 0,Y 326.595,Z 274.612,A -85,B 0,C 180,E1 -15052.788,E2 -15052.788} C_VEL
LIN {X 0,Y 326.68,Z 274.604,A -85,B 0,C 180,E1 -15055.484,E2 -15055.484} C_VEL
LIN {X 0,Y 326.669,Z 274.607,A -85,B 0,C 180,E1 -15059.657,E2 -15059.657} C_VEL
LIN {X 0,Y 326.681,Z 274.623,A -85,B 0,C 180,E1 -15060.427,E2 -15060.427} C_VEL
LIN {X 0,Y 326.917,Z 275.834,A -85,B 0,C 180,E1 -15060.806,E2 -15060.806} C_VEL
LIN {X 0,Y 329.72,Z 286.72,A -85,B 0,C 180,E1 -15061.208,E2 -15061.208} C_VEL
LIN {X 0,Y 331.391,Z 296.904,A -85,B 0,C 180,E1 -15061.535,E2 -15061.535} C_VEL
LIN {X 0,Y 330.271,Z 352.692,A -85,B 0,C 180,E1 -15062.907,E2 -15062.907} C_VEL
LIN {X 0,Y 329.958,Z 363.325,A -85,B 0,C 180,E1 -15063.352,E2 -15063.352} C_VEL
LIN {X 0,Y 329.467,Z 374.646,A -85,B 0,C 180,E1 -15064.069,E2 -15064.069} C_VEL
LIN {X 0,Y 328.942,Z 383.801,A -85,B 0,C 180,E1 -15064.861,E2 -15064.861} C_VEL
LIN {X 0,Y 328.537,Z 390.943,A -85,B 0,C 180,E1 -15065.623,E2 -15065.623} C_VEL
LIN {X 0,Y 327.914,Z 399.285,A -85,B 0,C 180,E1 -15066.718,E2 -15066.718} C_VEL
LIN {X 0,Y 327.222,Z 406.973,A -85,B 0,C 180,E1 -15067.958,E2 -15067.958} C_VEL
LIN {X 0,Y 326.678,Z 413.479,A -85,B 0,C 180,E1 -15069.244,E2 -15069.244} C_VEL
LIN {X 0,Y 326.244,Z 419.208,A -85,B 0,C 180,E1 -15070.629,E2 -15070.629} C_VEL
LIN {X 0,Y 325.757,Z 424.969,A -85,B 0,C 180,E1 -15072.373,E2 -15072.373} C_VEL
LIN {X 0,Y 325.488,Z 428.354,A -85,B 0,C 180,E1 -15073.704,E2 -15073.704} C_VEL
LIN {X 0,Y 325.132,Z 431.777,A -85,B 0,C 180,E1 -15075.504,E2 -15075.504} C_VEL
LIN {X 0,Y 324.902,Z 434.485,A -85,B 0,C 180,E1 -15077.891,E2 -15077.891} C_VEL
LIN {X 0,Y 324.95,Z 435.259,A -85,B 0,C 180,E1 -15079.548,E2 -15079.548} C_VEL
LIN {X 0,Y 325.082,Z 435.127,A -85,B 0,C 180,E1 -15081.176,E2 -15081.176} C_VEL
LIN {X 0,Y 325.404,Z 433.917,A -85,B 0,C 180,E1 -15083.044,E2 -15083.044} C_VEL
LIN {X 0,Y 325.765,Z 431.943,A -85,B 0,C 180,E1 -15084.573,E2 -15084.573} C_VEL
LIN {X 0,Y 325.376,Z 430.32,A -85,B 0,C 180,E1 -15085.571,E2 -15085.571} C_VEL
LIN {X 0,Y 323.073,Z 427.212,A -85,B 0,C 180,E1 -15087.191,E2 -15087.191} C_VEL
LIN {X 0,Y 320.915,Z 423.314,A -85,B 0,C 180,E1 -15088.768,E2 -15088.768} C_VEL
LIN {X 0,Y 320.749,Z 420.351,A -85,B 0,C 180,E1 -15089.681,E2 -15089.681} C_VEL
LIN {X 0,Y 321.689,Z 413.951,A -85,B 0,C 180,E1 -15091.274,E2 -15091.274} C_VEL
LIN {X 0,Y 322.894,Z 406.186,A -85,B 0,C 180,E1 -15092.803,E2 -15092.803} C_VEL
LIN {X 0,Y 324.033,Z 397.689,A -85,B 0,C 180,E1 -15094.121,E2 -15094.121} C_VEL
LIN {X 0,Y 325.002,Z 388.321,A -85,B 0,C 180,E1 -15095.259,E2 -15095.259} C_VEL
LIN {X 0,Y 325.735,Z 380.105,A -85,B 0,C 180,E1 -15096.054,E2 -15096.054} C_VEL
LIN {X 0,Y 326.466,Z 371.549,A -85,B 0,C 180,E1 -15096.7,E2 -15096.7} C_VEL
LIN {X 0,Y 326.93,Z 361.757,A -85,B 0,C 180,E1 -15097.265,E2 -15097.265} C_VEL
LIN {X 0,Y 327.355,Z 350.592,A -85,B 0,C 180,E1 -15097.686,E2 -15097.686} C_VEL
LIN {X 0,Y 328.706,Z 298.691,A -85,B 0,C 180,E1 -15099.016,E2 -15099.016} C_VEL
LIN {X 0,Y 325.048,Z 288.744,A -85,B 0,C 180,E1 -15099.618,E2 -15099.618} C_VEL
LIN {X 0,Y 320.056,Z 277.33,A -85,B 0,C 180,E1 -15100.433,E2 -15100.433} C_VEL
LIN {X 0,Y 319.704,Z 275.481,A -85,B 0,C 180,E1 -15101.113,E2 -15101.113} C_VEL
LIN {X 0,Y 319.722,Z 275.472,A -85,B 0,C 180,E1 -15105.277,E2 -15105.277} C_VEL
LIN {X 0,Y 319.744,Z 275.468,A -85,B 0,C 180,E1 -15109.874,E2 -15109.874} C_VEL
LIN {X 0,Y 319.905,Z 275.448,A -85,B 0,C 180,E1 -15112.427,E2 -15112.427} C_VEL
LIN {X 0,Y 319.741,Z 275.466,A -85,B 0,C 180,E1 -15114.957,E2 -15114.957} C_VEL
LIN {X 0,Y 319.984,Z 275.434,A -85,B 0,C 180,E1 -15117.483,E2 -15117.483} C_VEL
LIN {X 0,Y 320.142,Z 275.42,A -85,B 0,C 180,E1 -15120.001,E2 -15120.001} C_VEL
LIN {X 0,Y 319.984,Z 275.44,A -85,B 0,C 180,E1 -15122.519,E2 -15122.519} C_VEL
LIN {X 0,Y 319.944,Z 275.445,A -85,B 0,C 180,E1 -15126.307,E2 -15126.307} C_VEL
LIN {X 0,Y 319.836,Z 275.452,A -85,B 0,C 180,E1 -15128.849,E2 -15128.849} C_VEL
LIN {X 0,Y 319.674,Z 275.47,A -85,B 0,C 180,E1 -15132.701,E2 -15132.701} C_VEL
LIN {X 0,Y 319.693,Z 275.472,A -85,B 0,C 180,E1 -15135.297,E2 -15135.297} C_VEL
LIN {X 0,Y 319.669,Z 275.475,A -85,B 0,C 180,E1 -15139.256,E2 -15139.256} C_VEL
LIN {X 0,Y 319.565,Z 275.488,A -85,B 0,C 180,E1 -15143.321,E2 -15143.321} C_VEL
LIN {X 0,Y 319.63,Z 275.475,A -85,B 0,C 180,E1 -15146.089,E2 -15146.089} C_VEL
LIN {X 0,Y 319.585,Z 275.479,A -85,B 0,C 180,E1 -15148.935,E2 -15148.935} C_VEL
LIN {X 0,Y 319.528,Z 275.496,A -85,B 0,C 180,E1 -15151.863,E2 -15151.863} C_VEL
LIN {X 0,Y 319.576,Z 275.489,A -85,B 0,C 180,E1 -15155.544,E2 -15155.544} C_VEL
LIN {X 0,Y 319.579,Z 275.484,A -85,B 0,C 180,E1 -15158.008,E2 -15158.008} C_VEL
LIN {X 0,Y 319.569,Z 275.489,A -85,B 0,C 180,E1 -15161.607,E2 -15161.607} C_VEL
LIN {X 0,Y 319.519,Z 275.497,A -85,B 0,C 180,E1 -15165.264,E2 -15165.264} C_VEL
LIN {X 0,Y 319.527,Z 275.495,A -85,B 0,C 180,E1 -15168.713,E2 -15168.713} C_VEL
LIN {X 0,Y 319.577,Z 275.494,A -85,B 0,C 180,E1 -15172.345,E2 -15172.345} C_VEL
LIN {X 0,Y 319.56,Z 275.492,A -85,B 0,C 180,E1 -15175.125,E2 -15175.125} C_VEL
LIN {X 0,Y 319.566,Z 275.493,A -85,B 0,C 180,E1 -15179.06,E2 -15179.06} C_VEL
LIN {X 0,Y 319.631,Z 275.515,A -85,B 0,C 180,E1 -15179.553,E2 -15179.553} C_VEL
LIN {X 0,Y 321.933,Z 285.569,A -85,B 0,C 180,E1 -15182.714,E2 -15182.714} C_VEL
LIN {X 0,Y 323.098,Z 292.938,A -85,B 0,C 180,E1 -15184.903,E2 -15184.903} C_VEL
LIN {X 0,Y 321.594,Z 307.018,A -85,B 0,C 180,E1 -15188.646,E2 -15188.646} C_VEL
LIN {X 0,Y 321.591,Z 307.878,A -85,B 0,C 180,E1 -15188.797,E2 -15188.797} C_VEL
LIN {X 0,Y 325.065,Z 326.366,A -85,B 0,C 180,E1 -15189.629,E2 -15189.629} C_VEL
LIN {X 0,Y 327.264,Z 343.125,A -85,B 0,C 180,E1 -15190.275,E2 -15190.275} C_VEL
LIN {X 0,Y 327.671,Z 349.675,A -85,B 0,C 180,E1 -15190.485,E2 -15190.485} C_VEL
LIN {X 0,Y 326.566,Z 387.874,A -85,B 0,C 180,E1 -15191.485,E2 -15191.485} C_VEL
LIN {X 0,Y 325.807,Z 400.028,A -85,B 0,C 180,E1 -15192.031,E2 -15192.031} C_VEL
LIN {X 0,Y 324.878,Z 409.887,A -85,B 0,C 180,E1 -15192.696,E2 -15192.696} C_VEL
LIN {X 0,Y 323.927,Z 418.536,A -85,B 0,C 180,E1 -15193.456,E2 -15193.456} C_VEL
LIN {X 0,Y 322.861,Z 426.872,A -85,B 0,C 180,E1 -15194.373,E2 -15194.373} C_VEL
LIN {X 0,Y 321.828,Z 434.808,A -85,B 0,C 180,E1 -15195.456,E2 -15195.456} C_VEL
LIN {X 0,Y 320.763,Z 442.272,A -85,B 0,C 180,E1 -15196.7,E2 -15196.7} C_VEL
LIN {X 0,Y 319.781,Z 449.883,A -85,B 0,C 180,E1 -15198.271,E2 -15198.271} C_VEL
LIN {X 0,Y 318.929,Z 455.882,A -85,B 0,C 180,E1 -15199.847,E2 -15199.847} C_VEL
LIN {X 0,Y 318.502,Z 459.828,A -85,B 0,C 180,E1 -15201.115,E2 -15201.115} C_VEL
LIN {X 0,Y 318.08,Z 464.386,A -85,B 0,C 180,E1 -15203.02,E2 -15203.02} C_VEL
LIN {X 0,Y 317.914,Z 466.541,A -85,B 0,C 180,E1 -15204.158,E2 -15204.158} C_VEL
LIN {X 0,Y 317.912,Z 469.12,A -85,B 0,C 180,E1 -15206.198,E2 -15206.198} C_VEL
LIN {X 0,Y 317.871,Z 470.119,A -85,B 0,C 180,E1 -15207.466,E2 -15207.466} C_VEL
LIN {X 0,Y 317.961,Z 470.533,A -85,B 0,C 180,E1 -15208.734,E2 -15208.734} C_VEL
LIN {X 0,Y 318.11,Z 470.397,A -85,B 0,C 180,E1 -15210,E2 -15210} C_VEL
LIN {X 0,Y 318.014,Z 469.759,A -85,B 0,C 180,E1 -15211.267,E2 -15211.267} C_VEL
LIN {X 0,Y 317.917,Z 468.619,A -85,B 0,C 180,E1 -15212.534,E2 -15212.534} C_VEL
LIN {X 0,Y 317.969,Z 466.952,A -85,B 0,C 180,E1 -15213.802,E2 -15213.802} C_VEL
LIN {X 0,Y 317.906,Z 463.947,A -85,B 0,C 180,E1 -15215.399,E2 -15215.399} C_VEL
LIN {X 0,Y 318.103,Z 459.963,A -85,B 0,C 180,E1 -15216.98,E2 -15216.98} C_VEL
LIN {X 0,Y 318.394,Z 454.804,A -85,B 0,C 180,E1 -15218.569,E2 -15218.569} C_VEL
LIN {X 0,Y 318.677,Z 449.744,A -85,B 0,C 180,E1 -15219.841,E2 -15219.841} C_VEL
LIN {X 0,Y 319.221,Z 443.65,A -85,B 0,C 180,E1 -15221.107,E2 -15221.107} C_VEL
LIN {X 0,Y 319.845,Z 436.221,A -85,B 0,C 180,E1 -15222.371,E2 -15222.371} C_VEL
LIN {X 0,Y 320.532,Z 428.277,A -85,B 0,C 180,E1 -15223.472,E2 -15223.472} C_VEL
LIN {X 0,Y 321.269,Z 418.388,A -85,B 0,C 180,E1 -15224.571,E2 -15224.571} C_VEL
LIN {X 0,Y 322.111,Z 406.917,A -85,B 0,C 180,E1 -15225.502,E2 -15225.502} C_VEL
LIN {X 0,Y 322.698,Z 396.994,A -85,B 0,C 180,E1 -15226.081,E2 -15226.081} C_VEL
LIN {X 0,Y 323.102,Z 387.529,A -85,B 0,C 180,E1 -15226.46,E2 -15226.46} C_VEL
LIN {X 0,Y 323.756,Z 345.734,A -85,B 0,C 180,E1 -15227.523,E2 -15227.523} C_VEL
LIN {X 0,Y 320.017,Z 310.44,A -85,B 0,C 180,E1 -15228.61,E2 -15228.61} C_VEL
LIN {X 0,Y 321.288,Z 296.39,A -85,B 0,C 180,E1 -15232.507,E2 -15232.507} C_VEL
LIN {X 0,Y 321.99,Z 289.244,A -85,B 0,C 180,E1 -15234.501,E2 -15234.501} C_VEL
LIN {X 0,Y 320.828,Z 281.673,A -85,B 0,C 180,E1 -15236.735,E2 -15236.735} C_VEL
LIN {X 0,Y 319.681,Z 275.477,A -85,B 0,C 180,E1 -15238.617,E2 -15238.617} C_VEL
LIN {X 0,Y 319.532,Z 275.495,A -85,B 0,C 180,E1 -15241.861,E2 -15241.861} C_VEL
LIN {X 0,Y 319.582,Z 275.492,A -85,B 0,C 180,E1 -15245.542,E2 -15245.542} C_VEL
LIN {X 0,Y 319.575,Z 275.488,A -85,B 0,C 180,E1 -15248.007,E2 -15248.007} C_VEL
LIN {X 0,Y 319.552,Z 275.495,A -85,B 0,C 180,E1 -15251.601,E2 -15251.601} C_VEL
LIN {X 0,Y 319.488,Z 275.5,A -85,B 0,C 180,E1 -15255.256,E2 -15255.256} C_VEL
LIN {X 0,Y 319.528,Z 275.493,A -85,B 0,C 180,E1 -15258.711,E2 -15258.711} C_VEL
LIN {X 0,Y 319.561,Z 275.489,A -85,B 0,C 180,E1 -15262.347,E2 -15262.347} C_VEL
LIN {X 0,Y 319.559,Z 275.49,A -85,B 0,C 180,E1 -15265.122,E2 -15265.122} C_VEL
LIN {X 0,Y 319.569,Z 275.488,A -85,B 0,C 180,E1 -15269.057,E2 -15269.057} C_VEL
LIN {X 0,Y 319.607,Z 275.483,A -85,B 0,C 180,E1 -15272.497,E2 -15272.497} C_VEL
LIN {X 0,Y 319.603,Z 275.486,A -85,B 0,C 180,E1 -15275.303,E2 -15275.303} C_VEL
LIN {X 0,Y 319.595,Z 275.486,A -85,B 0,C 180,E1 -15278.047,E2 -15278.047} C_VEL
LIN {X 0,Y 319.687,Z 275.473,A -85,B 0,C 180,E1 -15280.961,E2 -15280.961} C_VEL
LIN {X 0,Y 319.728,Z 275.47,A -85,B 0,C 180,E1 -15285.275,E2 -15285.275} C_VEL
LIN {X 0,Y 319.749,Z 275.468,A -85,B 0,C 180,E1 -15289.872,E2 -15289.872} C_VEL
LIN {X 0,Y 319.909,Z 275.445,A -85,B 0,C 180,E1 -15292.425,E2 -15292.425} C_VEL
LIN {X 0,Y 319.742,Z 275.466,A -85,B 0,C 180,E1 -15294.955,E2 -15294.955} C_VEL
LIN {X 0,Y 319.987,Z 275.439,A -85,B 0,C 180,E1 -15297.481,E2 -15297.481} C_VEL
LIN {X 0,Y 320.145,Z 275.418,A -85,B 0,C 180,E1 -15299.999,E2 -15299.999} C_VEL
LIN {X 0,Y 319.987,Z 275.435,A -85,B 0,C 180,E1 -15302.517,E2 -15302.517} C_VEL
LIN {X 0,Y 319.925,Z 275.443,A -85,B 0,C 180,E1 -15306.67,E2 -15306.67} C_VEL
LIN {X 0,Y 319.754,Z 275.466,A -85,B 0,C 180,E1 -15310.126,E2 -15310.126} C_VEL
LIN {X 0,Y 319.725,Z 275.468,A -85,B 0,C 180,E1 -15314.723,E2 -15314.723} C_VEL
LIN {X 0,Y 319.685,Z 275.474,A -85,B 0,C 180,E1 -15319.038,E2 -15319.038} C_VEL
LIN {X 0,Y 319.564,Z 275.49,A -85,B 0,C 180,E1 -15323.318,E2 -15323.318} C_VEL
LIN {X 0,Y 319.627,Z 275.482,A -85,B 0,C 180,E1 -15326.087,E2 -15326.087} C_VEL
LIN {X 0,Y 319.581,Z 275.486,A -85,B 0,C 180,E1 -15328.933,E2 -15328.933} C_VEL
LIN {X 0,Y 319.525,Z 275.497,A -85,B 0,C 180,E1 -15331.861,E2 -15331.861} C_VEL
LIN {X 0,Y 319.573,Z 275.491,A -85,B 0,C 180,E1 -15335.542,E2 -15335.542} C_VEL
LIN {X 0,Y 319.591,Z 275.487,A -85,B 0,C 180,E1 -15338.004,E2 -15338.004} C_VEL
LIN {X 0,Y 319.564,Z 275.493,A -85,B 0,C 180,E1 -15341.606,E2 -15341.606} C_VEL
LIN {X 0,Y 319.58,Z 275.488,A -85,B 0,C 180,E1 -15345.274,E2 -15345.274} C_VEL
LIN {X 0,Y 319.572,Z 275.487,A -85,B 0,C 180,E1 -15348.719,E2 -15348.719} C_VEL
LIN {X 0,Y 319.59,Z 275.486,A -85,B 0,C 180,E1 -15352.339,E2 -15352.339} C_VEL
LIN {X 0,Y 319.552,Z 275.49,A -85,B 0,C 180,E1 -15355.123,E2 -15355.123} C_VEL
LIN {X 0,Y 319.562,Z 275.489,A -85,B 0,C 180,E1 -15359.058,E2 -15359.058} C_VEL
LIN {X 0,Y 319.6,Z 275.484,A -85,B 0,C 180,E1 -15362.498,E2 -15362.498} C_VEL
LIN {X 0,Y 319.597,Z 275.486,A -85,B 0,C 180,E1 -15365.304,E2 -15365.304} C_VEL
LIN {X 0,Y 319.589,Z 275.488,A -85,B 0,C 180,E1 -15368.047,E2 -15368.047} C_VEL
LIN {X 0,Y 319.681,Z 275.473,A -85,B 0,C 180,E1 -15370.962,E2 -15370.962} C_VEL
LIN {X 0,Y 319.723,Z 275.47,A -85,B 0,C 180,E1 -15375.276,E2 -15375.276} C_VEL
LIN {X 0,Y 319.75,Z 275.47,A -85,B 0,C 180,E1 -15379.872,E2 -15379.872} C_VEL
LIN {X 0,Y 319.924,Z 275.444,A -85,B 0,C 180,E1 -15382.426,E2 -15382.426} C_VEL
LIN {X 0,Y 319.736,Z 275.467,A -85,B 0,C 180,E1 -15384.956,E2 -15384.956} C_VEL
LIN {X 0,Y 319.98,Z 275.439,A -85,B 0,C 180,E1 -15387.482,E2 -15387.482} C_VEL
LIN {X 0,Y 320.142,Z 275.42,A -85,B 0,C 180,E1 -15390,E2 -15390} C_VEL
LIN {X 0,Y 319.981,Z 275.437,A -85,B 0,C 180,E1 -15392.517,E2 -15392.517} C_VEL
LIN {X 0,Y 319.936,Z 275.443,A -85,B 0,C 180,E1 -15396.305,E2 -15396.305} C_VEL
LIN {X 0,Y 319.834,Z 275.454,A -85,B 0,C 180,E1 -15398.848,E2 -15398.848} C_VEL
LIN {X 0,Y 319.675,Z 275.474,A -85,B 0,C 180,E1 -15402.7,E2 -15402.7} C_VEL
LIN {X 0,Y 319.69,Z 275.473,A -85,B 0,C 180,E1 -15405.295,E2 -15405.295} C_VEL
LIN {X 0,Y 319.664,Z 275.476,A -85,B 0,C 180,E1 -15409.255,E2 -15409.255} C_VEL
LIN {X 0,Y 319.552,Z 275.491,A -85,B 0,C 180,E1 -15413.32,E2 -15413.32} C_VEL
LIN {X 0,Y 319.624,Z 275.484,A -85,B 0,C 180,E1 -15416.088,E2 -15416.088} C_VEL
LIN {X 0,Y 319.656,Z 275.52,A -85,B 0,C 180,E1 -15420.284,E2 -15420.284} C_VEL
LIN {X 0,Y 319.787,Z 276.354,A -85,B 0,C 180,E1 -15420.492,E2 -15420.492} C_VEL
LIN {X 0,Y 322.913,Z 288.076,A -85,B 0,C 180,E1 -15420.942,E2 -15420.942} C_VEL
LIN {X 0,Y 324.496,Z 297.841,A -85,B 0,C 180,E1 -15421.263,E2 -15421.263} C_VEL
LIN {X 0,Y 323.329,Z 353.06,A -85,B 0,C 180,E1 -15422.654,E2 -15422.654} C_VEL
LIN {X 0,Y 323.016,Z 363.77,A -85,B 0,C 180,E1 -15423.113,E2 -15423.113} C_VEL
LIN {X 0,Y 322.486,Z 375.226,A -85,B 0,C 180,E1 -15423.858,E2 -15423.858} C_VEL
LIN {X 0,Y 321.936,Z 384.425,A -85,B 0,C 180,E1 -15424.676,E2 -15424.676} C_VEL
LIN {X 0,Y 321.425,Z 393.271,A -85,B 0,C 180,E1 -15425.676,E2 -15425.676} C_VEL
LIN {X 0,Y 320.828,Z 400.346,A -85,B 0,C 180,E1 -15426.649,E2 -15426.649} C_VEL
LIN {X 0,Y 320.207,Z 407.306,A -85,B 0,C 180,E1 -15427.804,E2 -15427.804} C_VEL
LIN {X 0,Y 319.753,Z 412.297,A -85,B 0,C 180,E1 -15428.785,E2 -15428.785} C_VEL
LIN {X 0,Y 319.35,Z 417.792,A -85,B 0,C 180,E1 -15430.068,E2 -15430.068} C_VEL
LIN {X 0,Y 318.832,Z 422.71,A -85,B 0,C 180,E1 -15431.459,E2 -15431.459} C_VEL
LIN {X 0,Y 318.546,Z 426.589,A -85,B 0,C 180,E1 -15432.809,E2 -15432.809} C_VEL
LIN {X 0,Y 318.297,Z 429.688,A -85,B 0,C 180,E1 -15434.146,E2 -15434.146} C_VEL
LIN {X 0,Y 317.987,Z 432.655,A -85,B 0,C 180,E1 -15435.879,E2 -15435.879} C_VEL
LIN {X 0,Y 317.885,Z 433.943,A -85,B 0,C 180,E1 -15436.85,E2 -15436.85} C_VEL
LIN {X 0,Y 317.811,Z 435.384,A -85,B 0,C 180,E1 -15438.751,E2 -15438.751} C_VEL
LIN {X 0,Y 317.947,Z 435.662,A -85,B 0,C 180,E1 -15440.681,E2 -15440.681} C_VEL
LIN {X 0,Y 318.08,Z 435.374,A -85,B 0,C 180,E1 -15441.783,E2 -15441.783} C_VEL
LIN {X 0,Y 318.419,Z 434.115,A -85,B 0,C 180,E1 -15443.423,E2 -15443.423} C_VEL
LIN {X 0,Y 318.827,Z 432.01,A -85,B 0,C 180,E1 -15445.033,E2 -15445.033} C_VEL
LIN {X 0,Y 319.419,Z 428.776,A -85,B 0,C 180,E1 -15446.727,E2 -15446.727} C_VEL
LIN {X 0,Y 320.311,Z 423.174,A -85,B 0,C 180,E1 -15448.835,E2 -15448.835} C_VEL
LIN {X 0,Y 320.749,Z 420.351,A -85,B 0,C 180,E1 -15449.681,E2 -15449.681} C_VEL
LIN {X 0,Y 320.614,Z 417.238,A -85,B 0,C 180,E1 -15450.565,E2 -15450.565} C_VEL
LIN {X 0,Y 318.696,Z 411.717,A -85,B 0,C 180,E1 -15452.003,E2 -15452.003} C_VEL
LIN {X 0,Y 316.9,Z 405.486,A -85,B 0,C 180,E1 -15453.368,E2 -15453.368} C_VEL
LIN {X 0,Y 316.901,Z 401.141,A -85,B 0,C 180,E1 -15454.099,E2 -15454.099} C_VEL
LIN {X 0,Y 318.064,Z 391.981,A -85,B 0,C 180,E1 -15455.352,E2 -15455.352} C_VEL
LIN {X 0,Y 319.115,Z 381.114,A -85,B 0,C 180,E1 -15456.475,E2 -15456.475} C_VEL
LIN {X 0,Y 319.946,Z 372.005,A -85,B 0,C 180,E1 -15457.183,E2 -15457.183} C_VEL
LIN {X 0,Y 320.393,Z 363.08,A -85,B 0,C 180,E1 -15457.719,E2 -15457.719} C_VEL
LIN {X 0,Y 320.782,Z 352.942,A -85,B 0,C 180,E1 -15458.134,E2 -15458.134} C_VEL
LIN {X 0,Y 322.459,Z 300.477,A -85,B 0,C 180,E1 -15459.509,E2 -15459.509} C_VEL
LIN {X 0,Y 317.009,Z 286.809,A -85,B 0,C 180,E1 -15460.409,E2 -15460.409} C_VEL
LIN {X 0,Y 313.035,Z 277.863,A -85,B 0,C 180,E1 -15461.094,E2 -15461.094} C_VEL
LIN {X 0,Y 312.651,Z 276.358,A -85,B 0,C 180,E1 -15461.659,E2 -15461.659} C_VEL
LIN {X 0,Y 312.685,Z 276.349,A -85,B 0,C 180,E1 -15465.687,E2 -15465.687} C_VEL
LIN {X 0,Y 312.69,Z 276.348,A -85,B 0,C 180,E1 -15469.643,E2 -15469.643} C_VEL
LIN {X 0,Y 312.846,Z 276.327,A -85,B 0,C 180,E1 -15472.255,E2 -15472.255} C_VEL
LIN {X 0,Y 312.711,Z 276.342,A -85,B 0,C 180,E1 -15474.843,E2 -15474.843} C_VEL
LIN {X 0,Y 312.983,Z 276.31,A -85,B 0,C 180,E1 -15478.714,E2 -15478.714} C_VEL
LIN {X 0,Y 312.985,Z 276.305,A -85,B 0,C 180,E1 -15481.288,E2 -15481.288} C_VEL
LIN {X 0,Y 312.711,Z 276.341,A -85,B 0,C 180,E1 -15485.159,E2 -15485.159} C_VEL
LIN {X 0,Y 312.865,Z 276.321,A -85,B 0,C 180,E1 -15487.747,E2 -15487.747} C_VEL
LIN {X 0,Y 312.662,Z 276.346,A -85,B 0,C 180,E1 -15491.673,E2 -15491.673} C_VEL
LIN {X 0,Y 312.694,Z 276.346,A -85,B 0,C 180,E1 -15494.889,E2 -15494.889} C_VEL
LIN {X 0,Y 312.625,Z 276.353,A -85,B 0,C 180,E1 -15499.238,E2 -15499.238} C_VEL
LIN {X 0,Y 312.541,Z 276.366,A -85,B 0,C 180,E1 -15502.79,E2 -15502.79} C_VEL
LIN {X 0,Y 312.579,Z 276.36,A -85,B 0,C 180,E1 -15506.724,E2 -15506.724} C_VEL
LIN {X 0,Y 312.541,Z 276.355,A -85,B 0,C 180,E1 -15509.651,E2 -15509.651} C_VEL
LIN {X 0,Y 312.516,Z 276.359,A -85,B 0,C 180,E1 -15513.69,E2 -15513.69} C_VEL
LIN {X 0,Y 312.538,Z 276.359,A -85,B 0,C 180,E1 -15517.384,E2 -15517.384} C_VEL
LIN {X 0,Y 312.499,Z 276.367,A -85,B 0,C 180,E1 -15520.709,E2 -15520.709} C_VEL
LIN {X 0,Y 312.515,Z 276.365,A -85,B 0,C 180,E1 -15524.199,E2 -15524.199} C_VEL
LIN {X 0,Y 312.484,Z 276.374,A -85,B 0,C 180,E1 -15527.92,E2 -15527.92} C_VEL
LIN {X 0,Y 312.535,Z 276.368,A -85,B 0,C 180,E1 -15531.912,E2 -15531.912} C_VEL
LIN {X 0,Y 312.506,Z 276.372,A -85,B 0,C 180,E1 -15535.791,E2 -15535.791} C_VEL
LIN {X 0,Y 312.554,Z 276.443,A -85,B 0,C 180,E1 -15538.999,E2 -15538.999} C_VEL
LIN {X 0,Y 314.971,Z 286.723,A -85,B 0,C 180,E1 -15542.356,E2 -15542.356} C_VEL
LIN {X 0,Y 316.245,Z 294.311,A -85,B 0,C 180,E1 -15544.673,E2 -15544.673} C_VEL
LIN {X 0,Y 314.834,Z 307.332,A -85,B 0,C 180,E1 -15548.165,E2 -15548.165} C_VEL
LIN {X 0,Y 318.585,Z 326.704,A -85,B 0,C 180,E1 -15549.077,E2 -15549.077} C_VEL
LIN {X 0,Y 320.874,Z 344.452,A -85,B 0,C 180,E1 -15549.787,E2 -15549.787} C_VEL
LIN {X 0,Y 321.187,Z 351.171,A -85,B 0,C 180,E1 -15550.004,E2 -15550.004} C_VEL
LIN {X 0,Y 320.026,Z 387.332,A -85,B 0,C 180,E1 -15550.976,E2 -15550.976} C_VEL
LIN {X 0,Y 319.308,Z 399.046,A -85,B 0,C 180,E1 -15551.507,E2 -15551.507} C_VEL
LIN {X 0,Y 318.353,Z 408.823,A -85,B 0,C 180,E1 -15552.164,E2 -15552.164} C_VEL
LIN {X 0,Y 317.331,Z 417.596,A -85,B 0,C 180,E1 -15552.936,E2 -15552.936} C_VEL
LIN {X 0,Y 316.24,Z 426.023,A -85,B 0,C 180,E1 -15553.872,E2 -15553.872} C_VEL
LIN {X 0,Y 315.148,Z 434.034,A -85,B 0,C 180,E1 -15554.975,E2 -15554.975} C_VEL
LIN {X 0,Y 314.079,Z 440.692,A -85,B 0,C 180,E1 -15556.082,E2 -15556.082} C_VEL
LIN {X 0,Y 313.19,Z 447.048,A -85,B 0,C 180,E1 -15557.363,E2 -15557.363} C_VEL
LIN {X 0,Y 312.416,Z 452.351,A -85,B 0,C 180,E1 -15558.649,E2 -15558.649} C_VEL
LIN {X 0,Y 311.675,Z 457.778,A -85,B 0,C 180,E1 -15560.264,E2 -15560.264} C_VEL
LIN {X 0,Y 311.124,Z 462.869,A -85,B 0,C 180,E1 -15562.211,E2 -15562.211} C_VEL
LIN {X 0,Y 310.83,Z 466.509,A -85,B 0,C 180,E1 -15564.192,E2 -15564.192} C_VEL
LIN {X 0,Y 310.816,Z 468.79,A -85,B 0,C 180,E1 -15566.111,E2 -15566.111} C_VEL
